RoboDK station: New Station (1).rdk

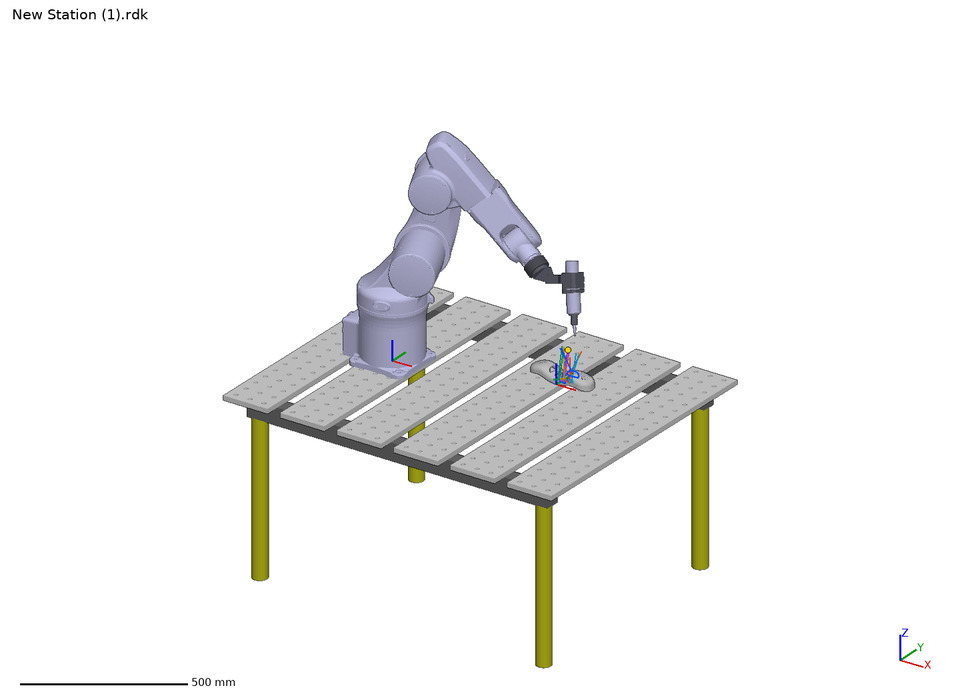
[picture v0: the station drawn from its stored meshes, robots at their saved joint values, targets as dots, program paths as lines]
Station New Station (1). Poses are relative to the parent item; angles as X-Y-Z fixed-axis rotations.
  - frame Adept Viper s650 Base at (-317.82, 0, 0) mm
    - robot Adept Viper s650: 6 axes, payload 5 kg, reach 653 mm, repeatability 0.02 mm, weight 28 kg
        modified DH rows (alpha deg, a mm, theta deg, d mm): 0, 0, 0, 335; -90, 75, 0, 0; 0, 270, -180, 0; -90, 90, 0, 295; 90, 0, 0, 0; -90, 0, 180, 80
        joint limits [-170, -190, -29, -190, -120, -360] to [170, 45, 256, 190, 120, 360]; home [0, -90, 180, 0, 0, 0]; saved at [24.912, -79.024, 220.131, -106.88, 32.598, 110.378]
      - tool Spindle, TCP at (32, 0, 260) mm, rotated rx 0 ry 39 rz 0 deg, size 157.3 x 72 x 259.9 mm
  - object Table at (0, 0, 0) mm, size 1193.8 x 965.2 x 609.6 mm, geometry from welding_table.sld
  - frame Deburring Frame at (278.6, 0, 88) mm
    - object telephone at (0, 0, 0) mm, rotated rx 0 ry 0 rz 90 deg, size 69.7 x 219.4 x 43.4 mm, geometry from telephone.stl
  - machining project telephone Settings: rotZ(0) | rotX(0)*rotY(0) | rotz(0) | onStart | onPathStart | onApproach | onPoint | onRetract | onFinish | SetRPM(%1) | SetTool(%1) | Extruder(%1) | default | default | OutOnMov(%1) | OutOffMov(%1) | onPathFinish | M_RunCode(%1)
  - machining project Path2 settings: rotZ(0) | rotX(0)*rotY(0) | rotz(0) | onStart | onPathStart | onApproach | onPoint | onRetract | onFinish | SetRPM(%1) | SetTool(%1) | Extruder(%1) | default | default | OutOnMov(%1) | OutOffMov(%1) | onPathFinish | M_RunCode(%1)
  - program Path2 (91 instructions, listed below)
  - machining project Path3 settings: rotZ(0) | rotX(0)*rotY(0) | rotz(0) | onStart | onPathStart | onApproach | onPoint | onRetract | onFinish | SetRPM(%1) | SetTool(%1) | Extruder(%1) | default | default | OutOnMov(%1) | OutOffMov(%1) | onPathFinish | M_RunCode(%1)
  - program Path3 (67 instructions, listed below)
  - machining project Path4 settings: rotZ(0) | rotX(0)*rotY(0) | rotz(0) | onStart | onPathStart | onApproach | onPoint | onRetract | onFinish | SetRPM(%1) | SetTool(%1) | Extruder(%1) | default | default | OutOnMov(%1) | OutOffMov(%1) | onPathFinish | M_RunCode(%1)
  - program Path4 (70 instructions, listed below)
  - machining project Path5 settings: rotZ(0) | rotX(0)*rotY(0) | rotz(0) | onStart | onPathStart | onApproach | onPoint | onRetract | onFinish | SetRPM(%1) | SetTool(%1) | Extruder(%1) | default | default | OutOnMov(%1) | OutOffMov(%1) | onPathFinish | M_RunCode(%1)
  - program Path5 (63 instructions, listed below)
  - machining project Path6 settings: rotZ(0) | rotX(0)*rotY(0) | rotz(0) | onStart | onPathStart | onApproach | onPoint | onRetract | onFinish | SetRPM(%1) | SetTool(%1) | Extruder(%1) | default | default | OutOnMov(%1) | OutOffMov(%1) | onPathFinish | M_RunCode(%1)
  - program Path6 (66 instructions, listed below)
  - machining project Path7 settings: rotZ(0) | rotX(0)*rotY(0) | rotz(0) | onStart | onPathStart | onApproach | onPoint | onRetract | onFinish | SetRPM(%1) | SetTool(%1) | Extruder(%1) | default | default | OutOnMov(%1) | OutOffMov(%1) | onPathFinish | M_RunCode(%1)
  - program Path7 (67 instructions, listed below)
  - program telephone (90 instructions, listed below)
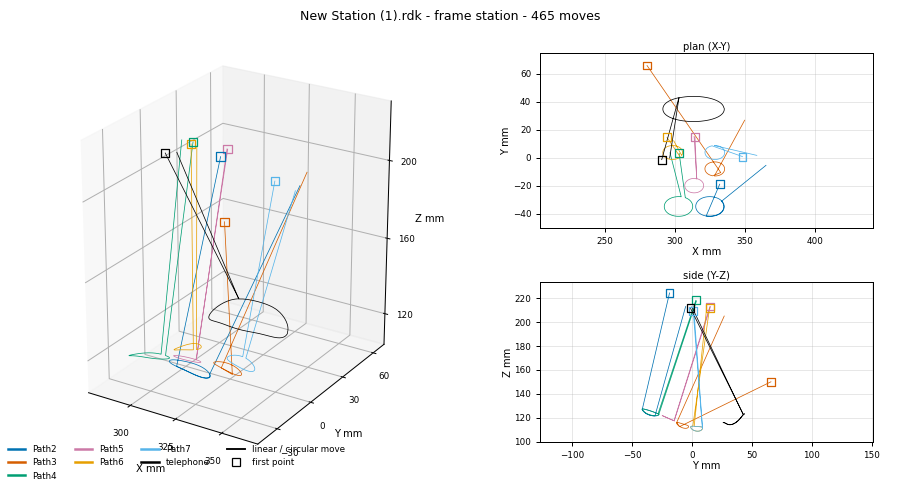
[picture p0: tool path of New Station (1).rdk in frame station, 465 of 465 moves have a stored position in this frame; points joined in program order, loops and branches not executed]

--- program Path2 (robot Adept Viper s650) ---
  Smooth(1)
  Set speed (1000.0 mm/s)
  Set Ref.: Deburring Frame
  Set Tool: Spindle
  Show Spindle
  MoveJ 1 to (53.51, -18.8, 136.35) mm, rotated rx -174.16 ry 13.06 rz 91.32 deg; joints [11.822, -84.058, 219.35, -116.51, 14.318, 120.131]
  MoveL 2 to (53.51, -18.8, 136.35) mm, rotated rx -174.16 ry 13.06 rz 91.32 deg; joints [11.822, -84.058, 219.35, -116.51, 14.318, 120.131]
  MoveL 3 to (43.86, -41.5, 39.44) mm, rotated rx -174.16 ry 13.06 rz 91.32 deg; joints [9.776, -66.741, 219.947, -154.659, 26.957, 158.699]
  MoveL 4 to (43.86, -41.5, 39.44) mm, rotated rx -174.16 ry 13.06 rz 91.32 deg; joints [9.776, -66.741, 219.947, -154.659, 26.957, 158.699]
  Set speed (50.0 mm/s)
  MoveL 5 to (45.33, -41.69, 39.33) mm, rotated rx -172.97 ry 12.9 rz 91.58 deg; joints [10.651, -66.44, 219.515, -151.515, 27.179, 155.489]
  MoveL 6 to (46.59, -41.73, 39.17) mm, rotated rx -170.38 ry 12.62 rz 92.12 deg; joints [12.268, -65.809, 218.773, -145.586, 28.019, 149.205]
  MoveL 7 to (48.09, -41.66, 38.87) mm, rotated rx -167.49 ry 12.41 rz 92.73 deg; joints [14.064, -64.95, 218.023, -139.796, 29.5, 143.03]
  MoveL 8 to (49.56, -41.44, 38.46) mm, rotated rx -164.73 ry 12.23 rz 93.31 deg; joints [15.752, -63.993, 217.309, -135.006, 31.231, 137.876]
  MoveL 9 to (50.68, -41.18, 38.07) mm, rotated rx -162.31 ry 12.13 rz 93.84 deg; joints [17.177, -63.064, 216.743, -131.537, 33, 134.068]
  MoveL 10 to (52.03, -40.71, 37.51) mm, rotated rx -160 ry 12.1 rz 94.36 deg; joints [18.544, -62.081, 216.284, -128.828, 34.916, 131.079]
  MoveL 11 to (53.28, -40.1, 36.89) mm, rotated rx -158.2 ry 12.02 rz 94.76 deg; joints [19.627, -61.249, 215.866, -126.779, 36.409, 128.843]
  MoveL 12 to (53.74, -39.81, 36.63) mm, rotated rx -157.25 ry 11.99 rz 94.98 deg; joints [20.161, -60.808, 215.677, -125.878, 37.231, 127.818]
  MoveL 13 to (54.69, -39.07, 36.05) mm, rotated rx -156.81 ry 12.12 rz 95.14 deg; joints [20.524, -60.571, 215.832, -125.816, 37.899, 127.837]
  MoveL 14 to (55.47, -38.25, 35.52) mm, rotated rx -156.78 ry 12.34 rz 95.24 deg; joints [20.662, -60.55, 216.211, -126.356, 38.326, 128.538]
  MoveL 15 to (55.93, -37.57, 35.15) mm, rotated rx -157.12 ry 12.6 rz 95.26 deg; joints [20.578, -60.709, 216.714, -127.342, 38.499, 129.714]
  MoveL 16 to (56.35, -36.71, 34.75) mm, rotated rx -157.66 ry 12.9 rz 95.24 deg; joints [20.401, -60.973, 217.335, -128.582, 38.581, 131.196]
  MoveL 17 to (56.4, -36.58, 34.7) mm, rotated rx -158.04 ry 13.08 rz 95.22 deg; joints [20.221, -61.139, 217.652, -129.392, 38.555, 132.109]
  MoveL 18 to (56.62, -35.75, 34.39) mm, rotated rx -158.41 ry 13.23 rz 95.18 deg; joints [20.104, -61.343, 218.07, -130.132, 38.577, 133.023]
  MoveL 19 to (56.71, -34.89, 34.12) mm, rotated rx -159.01 ry 13.46 rz 95.1 deg; joints [19.853, -61.655, 218.636, -131.298, 38.533, 134.398]
  MoveL 20 to (56.68, -34.23, 33.95) mm, rotated rx -159.47 ry 13.6 rz 95.03 deg; joints [19.65, -61.902, 219.035, -132.122, 38.457, 135.366]
  MoveL 21 to (56.63, -33.9, 33.88) mm, rotated rx -159.71 ry 13.68 rz 95 deg; joints [19.537, -62.031, 219.25, -132.577, 38.428, 135.892]
  MoveL 22 to (56.44, -33.13, 33.73) mm, rotated rx -159.89 ry 13.75 rz 94.97 deg; joints [19.455, -62.189, 219.552, -133.002, 38.469, 136.39]
  MoveL 23 to (56.13, -32.37, 33.63) mm, rotated rx -160.06 ry 13.79 rz 94.94 deg; joints [19.365, -62.356, 219.834, -133.373, 38.48, 136.815]
  MoveL 24 to (56.07, -32.27, 33.62) mm, rotated rx -160.12 ry 13.83 rz 94.94 deg; joints [19.327, -62.396, 219.921, -133.552, 38.502, 137.012]
  MoveL 25 to (55.61, -31.52, 33.57) mm, rotated rx -160.19 ry 13.93 rz 94.96 deg; joints [19.262, -62.53, 220.248, -133.964, 38.66, 137.442]
  MoveL 26 to (55, -30.79, 33.58) mm, rotated rx -160.3 ry 14.06 rz 94.97 deg; joints [19.152, -62.691, 220.623, -134.513, 38.828, 137.999]
  MoveL 27 to (54.88, -30.66, 33.59) mm, rotated rx -160.47 ry 14.24 rz 94.99 deg; joints [19.047, -62.763, 220.887, -135.12, 38.995, 138.642]
  MoveL 28 to (54.02, -29.92, 33.67) mm, rotated rx -160.96 ry 14.61 rz 94.98 deg; joints [18.699, -63.064, 221.608, -136.63, 39.279, 140.214]
  MoveL 29 to (53.03, -29.28, 33.8) mm, rotated rx -161.94 ry 15.12 rz 94.86 deg; joints [18.069, -63.52, 222.542, -138.962, 39.476, 142.68]
  MoveL 30 to (52.23, -28.87, 33.92) mm, rotated rx -163.91 ry 15.86 rz 94.51 deg; joints [16.933, -64.207, 223.779, -142.808, 39.497, 146.856]
  MoveL 31 to (50.89, -28.36, 34.12) mm, rotated rx -166.32 ry 16.57 rz 93.97 deg; joints [15.492, -64.991, 225.06, -147.237, 39.413, 151.619]
  MoveL 32 to (49.47, -27.98, 34.33) mm, rotated rx -168.54 ry 17.08 rz 93.41 deg; joints [14.119, -65.637, 226.045, -151.185, 39.278, 155.822]
  MoveL 33 to (48.32, -27.79, 34.5) mm, rotated rx -170.84 ry 17.46 rz 92.77 deg; joints [12.719, -66.194, 226.83, -155.099, 39.06, 160.014]
  MoveL 34 to (46.67, -27.67, 34.72) mm, rotated rx -172.86 ry 17.76 rz 92.19 deg; joints [11.384, -66.632, 227.471, -158.665, 38.953, 163.726]
  MoveL 35 to (45, -27.73, 34.92) mm, rotated rx -174.72 ry 17.95 rz 91.63 deg; joints [10.113, -66.972, 227.927, -161.947, 38.808, 167.106]
  MoveL 36 to (43.78, -27.89, 35.08) mm, rotated rx -175.97 ry 18.12 rz 91.25 deg; joints [9.236, -67.133, 228.219, -164.217, 38.847, 169.427]
  MoveL 37 to (42.27, -28.24, 35.29) mm, rotated rx -176.64 ry 18.23 rz 91.05 deg; joints [8.625, -67.201, 228.359, -165.629, 38.902, 170.747]
  MoveL 38 to (40.89, -28.75, 35.53) mm, rotated rx -176.95 ry 18.33 rz 90.96 deg; joints [8.228, -67.202, 228.406, -166.445, 38.983, 171.424]
  MoveL 39 to (40.41, -28.98, 35.63) mm, rotated rx -176.9 ry 18.46 rz 90.98 deg; joints [8.178, -67.138, 228.477, -166.546, 39.248, 171.458]
  MoveL 40 to (39.33, -29.62, 35.89) mm, rotated rx -176.68 ry 18.53 rz 91.06 deg; joints [8.118, -67.068, 228.403, -166.466, 39.328, 171.186]
  MoveL 41 to (38.41, -30.35, 36.19) mm, rotated rx -176.39 ry 18.62 rz 91.15 deg; joints [8.116, -66.969, 228.315, -166.271, 39.458, 170.807]
  MoveL 42 to (37.75, -31.04, 36.46) mm, rotated rx -176.1 ry 18.66 rz 91.25 deg; joints [8.158, -66.887, 228.182, -165.98, 39.479, 170.362]
  MoveL 43 to (37.17, -31.88, 36.78) mm, rotated rx -175.9 ry 18.66 rz 91.31 deg; joints [8.155, -66.817, 227.997, -165.796, 39.392, 170.041]
  MoveL 44 to (36.78, -32.66, 37.08) mm, rotated rx -175.77 ry 18.64 rz 91.35 deg; joints [8.146, -66.765, 227.798, -165.657, 39.238, 169.804]
  MoveL 45 to (36.52, -33.55, 37.4) mm, rotated rx -175.73 ry 18.58 rz 91.36 deg; joints [8.107, -66.726, 227.548, -165.591, 38.975, 169.662]
  MoveL 46 to (36.49, -33.71, 37.46) mm, rotated rx -175.79 ry 18.46 rz 91.34 deg; joints [8.064, -66.767, 227.422, -165.611, 38.691, 169.675]
  MoveL 47 to (36.4, -34.56, 37.75) mm, rotated rx -175.86 ry 18.36 rz 91.31 deg; joints [7.995, -66.754, 227.145, -165.641, 38.319, 169.671]
  MoveL 48 to (36.44, -35.26, 37.98) mm, rotated rx -175.93 ry 18.22 rz 91.27 deg; joints [7.945, -66.757, 226.875, -165.64, 37.909, 169.657]
  MoveL 49 to (36.47, -35.43, 38.03) mm, rotated rx -176.04 ry 18.04 rz 91.23 deg; joints [7.883, -66.824, 226.687, -165.674, 37.464, 169.694]
  MoveL 50 to (36.55, -35.87, 38.17) mm, rotated rx -176.16 ry 17.8 rz 91.18 deg; joints [7.816, -66.884, 226.382, -165.673, 36.854, 169.695]
  MoveL 51 to (36.82, -36.7, 38.42) mm, rotated rx -176.39 ry 17.5 rz 91.09 deg; joints [7.705, -66.933, 225.94, -165.772, 36.048, 169.825]
  MoveL 52 to (37.24, -37.52, 38.65) mm, rotated rx -176.52 ry 17.21 rz 91.03 deg; joints [7.676, -66.954, 225.493, -165.673, 35.297, 169.756]
  MoveL 53 to (37.33, -37.66, 38.69) mm, rotated rx -176.89 ry 16.75 rz 90.9 deg; joints [7.471, -67.114, 225.075, -165.954, 34.228, 170.077]
  MoveL 54 to (37.95, -38.47, 38.91) mm, rotated rx -177.09 ry 16.38 rz 90.82 deg; joints [7.424, -67.143, 224.535, -165.89, 33.278, 170.077]
  MoveL 55 to (38.7, -39.22, 39.09) mm, rotated rx -177.32 ry 15.94 rz 90.74 deg; joints [7.382, -67.179, 223.946, -165.795, 32.213, 170.065]
  MoveL 56 to (39.08, -39.52, 39.16) mm, rotated rx -177.53 ry 15.3 rz 90.65 deg; joints [7.288, -67.295, 223.269, -165.625, 30.785, 169.925]
  MoveL 57 to (40.1, -40.19, 39.3) mm, rotated rx -177.34 ry 14.81 rz 90.68 deg; joints [7.513, -67.265, 222.578, -164.583, 29.711, 168.919]
  MoveL 58 to (41.24, -40.74, 39.4) mm, rotated rx -176.81 ry 14.17 rz 90.78 deg; joints [7.947, -67.204, 221.704, -162.55, 28.426, 166.864]
  MoveL 59 to (42.44, -41.17, 39.45) mm, rotated rx -175.65 ry 13.56 rz 91.02 deg; joints [8.749, -67.031, 220.797, -159.011, 27.45, 163.202]
  MoveL 60 to (43.86, -41.5, 39.44) mm, rotated rx -173.92 ry 13.08 rz 91.38 deg; joints [9.914, -66.696, 219.942, -154.19, 27.101, 158.188]
  MoveL 61 to (45.34, -41.52, 39.29) mm, rotated rx -171.6 ry 12.58 rz 91.84 deg; joints [11.422, -66.186, 219.018, -148.104, 27.266, 151.813]
  MoveL 62 to (46.58, -41.56, 39.13) mm, rotated rx -168.9 ry 12.22 rz 92.38 deg; joints [13.088, -65.46, 218.138, -141.952, 28.204, 145.277]
  MoveL 63 to (48.06, -41.49, 38.83) mm, rotated rx -166.24 ry 11.93 rz 92.9 deg; joints [14.75, -64.594, 217.31, -136.578, 29.594, 139.553]
  MoveL 64 to (49.51, -41.27, 38.43) mm, rotated rx -163.53 ry 11.65 rz 93.42 deg; joints [16.398, -63.592, 216.465, -131.819, 31.279, 134.431]
  MoveL 65 to (50.62, -41, 38.05) mm, rotated rx -161.08 ry 11.6 rz 93.94 deg; joints [17.825, -62.605, 215.925, -128.66, 33.238, 130.925]
  MoveL 66 to (51.95, -40.53, 37.5) mm, rotated rx -159.3 ry 11.65 rz 94.36 deg; joints [18.915, -61.802, 215.641, -126.857, 34.889, 128.946]
  MoveL 67 to (53.17, -39.92, 36.89) mm, rotated rx -157.83 ry 11.77 rz 94.75 deg; joints [19.816, -61.109, 215.54, -125.785, 36.408, 127.762]
  MoveL 68 to (53.63, -39.64, 36.64) mm, rotated rx -157.19 ry 12.16 rz 95.06 deg; joints [20.172, -60.818, 215.916, -126.318, 37.502, 128.254]
  MoveL 69 to (54.55, -38.91, 36.07) mm, rotated rx -157.07 ry 12.45 rz 95.21 deg; joints [20.369, -60.726, 216.335, -126.963, 38.124, 129.049]
  MoveL 70 to (55.3, -38.1, 35.55) mm, rotated rx -157.35 ry 12.89 rz 95.32 deg; joints [20.343, -60.835, 217.027, -128.315, 38.604, 130.633]
  MoveL 71 to (55.75, -37.44, 35.19) mm, rotated rx -157.59 ry 13.07 rz 95.33 deg; joints [20.309, -60.941, 217.398, -128.977, 38.761, 131.455]
  MoveL 72 to (56.15, -36.6, 34.8) mm, rotated rx -158.25 ry 13.39 rz 95.28 deg; joints [20.064, -61.246, 218.061, -130.387, 38.805, 133.132]
  MoveL 73 to (56.19, -36.48, 34.75) mm, rotated rx -158.63 ry 13.46 rz 95.21 deg; joints [19.891, -61.408, 218.241, -130.907, 38.632, 133.747]
  MoveL 74 to (56.4, -35.68, 34.45) mm, rotated rx -159.14 ry 13.62 rz 95.13 deg; joints [19.698, -61.665, 218.69, -131.811, 38.568, 134.849]
  MoveL 75 to (56.47, -34.86, 34.2) mm, rotated rx -159.52 ry 13.7 rz 95.05 deg; joints [19.559, -61.883, 219.034, -132.412, 38.492, 135.601]
  MoveL 76 to (56.44, -34.23, 34.04) mm, rotated rx -159.82 ry 13.74 rz 94.99 deg; joints [19.439, -62.062, 219.279, -132.837, 38.392, 136.129]
  MoveL 77 to (56.4, -33.92, 33.96) mm, rotated rx -159.94 ry 13.76 rz 94.96 deg; joints [19.387, -62.143, 219.405, -133.043, 38.37, 136.378]
  MoveL 78 to (56.21, -33.19, 33.83) mm, rotated rx -160.06 ry 13.79 rz 94.94 deg; joints [19.335, -62.276, 219.638, -133.302, 38.388, 136.694]
  MoveL 79 to (55.91, -32.47, 33.73) mm, rotated rx -160.13 ry 13.82 rz 94.94 deg; joints [19.294, -62.398, 219.877, -133.542, 38.452, 136.967]
  MoveL 80 to (55.86, -32.37, 33.72) mm, rotated rx -160.19 ry 13.91 rz 94.95 deg; joints [19.258, -62.429, 220.008, -133.814, 38.546, 137.257]
  MoveL 81 to (55.42, -31.65, 33.68) mm, rotated rx -160.15 ry 13.86 rz 94.94 deg; joints [19.251, -62.532, 220.147, -133.779, 38.549, 137.212]
  MoveL 82 to (54.83, -30.95, 33.69) mm, rotated rx -160.25 ry 14 rz 94.96 deg; joints [19.147, -62.684, 220.52, -134.331, 38.732, 137.772]
  Set speed (1000.0 mm/s)
  MoveL 83 to (54.83, -30.95, 33.69) mm, rotated rx -160.25 ry 14 rz 94.96 deg; joints [19.147, -62.684, 220.52, -134.331, 38.732, 137.772]
  MoveL 84 to (86.53, -5.35, 125.01) mm, rotated rx -160.25 ry 14 rz 94.96 deg; joints [24.912, -79.024, 220.131, -106.88, 32.598, 110.378]

--- program Path3 (robot Adept Viper s650) ---
  Smooth(1)
  Set speed (1000.0 mm/s)
  Set Ref.: Deburring Frame
  Set Tool: Spindle
  Show Spindle
  MoveJ 1 to (1.67, 65.89, 62.11) mm, rotated rx 112.25 ry 7.94 rz 37.78 deg; joints [0.056, -47.226, 255.354, -174.919, 106.228, -108.091]
  MoveL 2 to (1.67, 65.89, 62.11) mm, rotated rx 112.25 ry 7.94 rz 37.78 deg; joints [0.056, -47.226, 255.354, -174.919, 106.228, -108.091]
  MoveL 3 to (54.24, -10.47, 24.61) mm, rotated rx 114.73 ry 26.32 rz 46.09 deg; joints [4.762, -22.597, 229.967, -175.784, 116.598, -123.556]
  MoveL 4 to (54.24, -10.47, 24.61) mm, rotated rx 114.73 ry 26.32 rz 46.09 deg; joints [4.762, -22.597, 229.967, -175.784, 116.598, -123.556]
  Set speed (50.0 mm/s)
  MoveL 5 to (48.57, -12.8, 28.08) mm, rotated rx 159.78 ry 39.33 rz 76.86 deg; joints [5.018, -40.691, 237.454, -177.659, 97.243, -163.59]
  MoveL 6 to (47.94, -12.67, 28.14) mm, rotated rx -169.03 ry 22.67 rz 94.27 deg; joints [14.025, -63.487, 233.835, -158.545, 53.468, -195.376]
  MoveL 7 to (46.89, -12.37, 28.19) mm, rotated rx -170.53 ry 22.4 rz 93.64 deg; joints [13.125, -64.139, 233.981, -160.07, 52.42, -193.816]
  MoveL 8 to (45.93, -11.96, 28.15) mm, rotated rx -171.82 ry 22.21 rz 93.11 deg; joints [12.327, -64.636, 234.159, -161.496, 51.69, -192.362]
  MoveL 9 to (45.4, -11.66, 28.09) mm, rotated rx -172.72 ry 21.92 rz 92.73 deg; joints [11.785, -65.072, 234.167, -162.404, 50.838, -191.437]
  MoveL 10 to (44.66, -11.13, 27.96) mm, rotated rx -173.43 ry 21.4 rz 92.41 deg; joints [11.309, -65.625, 234.055, -163.035, 49.58, -190.865]
  MoveL 11 to (44.05, -10.53, 27.79) mm, rotated rx -173.69 ry 21.02 rz 92.27 deg; joints [11.086, -65.986, 233.978, -163.23, 48.738, -190.746]
  MoveL 12 to (43.98, -10.45, 27.76) mm, rotated rx -173.82 ry 20.62 rz 92.18 deg; joints [11.001, -66.278, 233.741, -163.162, 47.822, -190.853]
  MoveL 13 to (43.54, -9.83, 27.58) mm, rotated rx -173.99 ry 19.92 rz 92.06 deg; joints [10.851, -66.801, 233.402, -163.006, 46.272, -191.11]
  MoveL 14 to (43.23, -9.2, 27.38) mm, rotated rx -173.95 ry 19.13 rz 91.99 deg; joints [10.829, -67.302, 232.956, -162.489, 44.597, -191.739]
  MoveL 15 to (43.12, -8.87, 27.28) mm, rotated rx -173.82 ry 18.39 rz 91.96 deg; joints [10.883, -67.702, 232.44, -161.795, 43.026, -192.532]
  MoveL 16 to (43, -8.29, 27.1) mm, rotated rx -173.76 ry 17.72 rz 91.91 deg; joints [10.901, -68.066, 232.024, -161.223, 41.643, -193.173]
  MoveL 17 to (42.99, -8.22, 27.08) mm, rotated rx -173.72 ry 17.09 rz 91.85 deg; joints [10.914, -68.35, 231.513, -160.634, 40.291, -193.832]
  MoveL 18 to (42.97, -7.57, 26.89) mm, rotated rx -173.66 ry 16.35 rz 91.79 deg; joints [10.954, -68.699, 231.002, -159.866, 38.769, -194.658]
  MoveL 19 to (43, -7.34, 26.82) mm, rotated rx -173.54 ry 15.47 rz 91.73 deg; joints [11.013, -69.014, 230.257, -158.807, 36.96, -195.804]
  MoveL 20 to (43.14, -6.69, 26.62) mm, rotated rx -173.44 ry 14.52 rz 91.65 deg; joints [11.092, -69.343, 229.503, -157.566, 35.068, -197.1]
  MoveL 21 to (43.26, -6.34, 26.52) mm, rotated rx -173.43 ry 13.67 rz 91.56 deg; joints [11.105, -69.589, 228.762, -156.484, 33.356, -198.232]
  MoveL 22 to (43.42, -6.01, 26.42) mm, rotated rx -173.23 ry 12.74 rz 91.5 deg; joints [11.231, -69.768, 227.887, -154.819, 31.582, -199.964]
  MoveL 23 to (43.83, -5.37, 26.23) mm, rotated rx -172.99 ry 11.59 rz 91.42 deg; joints [11.426, -69.939, 226.791, -152.439, 29.459, -202.387]
  MoveL 24 to (44.3, -4.85, 26.08) mm, rotated rx -172.66 ry 10.38 rz 91.33 deg; joints [11.673, -70.003, 225.556, -149.424, 27.361, -205.452]
  MoveL 25 to (45.04, -4.25, 25.87) mm, rotated rx -172.01 ry 9.21 rz 91.29 deg; joints [12.166, -69.908, 224.264, -145.251, 25.634, -209.656]
  MoveL 26 to (46, -3.7, 25.65) mm, rotated rx -170.97 ry 8.3 rz 91.31 deg; joints [12.945, -69.621, 223.122, -140.355, 24.772, -214.564]
  MoveL 27 to (47.09, -3.29, 25.4) mm, rotated rx -169.51 ry 7.77 rz 91.43 deg; joints [14.016, -69.147, 222.263, -135.475, 25.003, -219.447]
  MoveL 28 to (48.28, -3.01, 25.13) mm, rotated rx -168.12 ry 7.6 rz 91.59 deg; joints [15.066, -68.635, 221.773, -132.011, 25.886, -222.878]
  MoveL 29 to (48.69, -2.95, 25.03) mm, rotated rx -166.9 ry 7.58 rz 91.76 deg; joints [15.877, -68.19, 221.477, -129.723, 26.848, -225.215]
  MoveL 30 to (49.99, -2.87, 24.7) mm, rotated rx -165.32 ry 7.68 rz 92.01 deg; joints [17.032, -67.511, 221.164, -127.27, 28.358, -227.631]
  MoveL 31 to (51.3, -2.96, 24.36) mm, rotated rx -163.86 ry 7.75 rz 92.23 deg; joints [18.081, -66.804, 220.793, -125.187, 29.751, -229.681]
  MoveL 32 to (51.51, -2.99, 24.3) mm, rotated rx -162.89 ry 7.95 rz 92.44 deg; joints [18.688, -66.388, 220.771, -124.486, 30.853, -230.431]
  MoveL 33 to (52.65, -3.23, 23.98) mm, rotated rx -161.8 ry 8.4 rz 92.75 deg; joints [19.468, -65.805, 220.907, -124.353, 32.414, -230.505]
  MoveL 34 to (53.7, -3.6, 23.69) mm, rotated rx -160.98 ry 8.89 rz 93.05 deg; joints [20.071, -65.303, 221.113, -124.641, 33.782, -230.153]
  MoveL 35 to (54.6, -4.06, 23.46) mm, rotated rx -160.88 ry 9.51 rz 93.28 deg; joints [20.231, -65.126, 221.659, -126.158, 34.719, -228.513]
  MoveL 36 to (55.29, -4.55, 23.32) mm, rotated rx -161.28 ry 10.32 rz 93.47 deg; joints [20.082, -65.172, 222.532, -128.668, 35.524, -225.839]
  MoveL 37 to (55.85, -5.07, 23.25) mm, rotated rx -161.89 ry 11.28 rz 93.66 deg; joints [19.794, -65.273, 223.605, -131.718, 36.473, -222.604]
  MoveL 38 to (56.26, -5.59, 23.24) mm, rotated rx -162.44 ry 12.21 rz 93.83 deg; joints [19.517, -65.315, 224.598, -134.473, 37.506, -219.687]
  MoveL 39 to (56.43, -5.85, 23.25) mm, rotated rx -162.79 ry 12.91 rz 93.96 deg; joints [19.325, -65.315, 225.357, -136.425, 38.407, -217.623]
  MoveL 40 to (56.58, -6.14, 23.28) mm, rotated rx -163.04 ry 13.52 rz 94.08 deg; joints [19.188, -65.26, 225.969, -137.968, 39.257, -215.992]
  MoveL 41 to (56.72, -6.44, 23.32) mm, rotated rx -163.24 ry 14.15 rz 94.21 deg; joints [19.068, -65.164, 226.573, -139.433, 40.195, -214.442]
  MoveL 42 to (56.82, -6.72, 23.37) mm, rotated rx -163.39 ry 14.76 rz 94.35 deg; joints [18.974, -65.031, 227.139, -140.743, 41.17, -213.057]
  MoveL 43 to (56.9, -7.01, 23.43) mm, rotated rx -163.49 ry 15.5 rz 94.53 deg; joints [18.894, -64.824, 227.799, -142.166, 42.424, -211.552]
  MoveL 44 to (57, -7.59, 23.59) mm, rotated rx -163.51 ry 16.29 rz 94.75 deg; joints [18.841, -64.511, 228.408, -143.494, 43.829, -210.165]
  MoveL 45 to (57.01, -7.75, 23.64) mm, rotated rx -163.42 ry 16.99 rz 94.97 deg; joints [18.85, -64.196, 228.988, -144.521, 45.2, -209.08]
  MoveL 46 to (56.99, -8.37, 23.85) mm, rotated rx -163.16 ry 17.86 rz 95.3 deg; joints [18.902, -63.694, 229.564, -145.553, 46.938, -208.031]
  MoveL 47 to (56.85, -9.04, 24.13) mm, rotated rx -162.67 ry 18.83 rz 95.75 deg; joints [19.031, -63.017, 230.154, -146.464, 49.031, -207.148]
  MoveL 48 to (56.6, -9.7, 24.46) mm, rotated rx -162.18 ry 19.49 rz 96.12 deg; joints [19.143, -62.477, 230.489, -146.953, 50.528, -206.742]
  MoveL 49 to (56.56, -9.79, 24.51) mm, rotated rx -161.62 ry 20.09 rz 96.51 deg; joints [19.35, -61.916, 230.84, -147.241, 52.027, -206.476]
  MoveL 50 to (56.1, -10.5, 24.94) mm, rotated rx -161.02 ry 20.74 rz 96.94 deg; joints [19.451, -61.321, 231.121, -147.636, 53.544, -206.229]
  MoveL 51 to (55.46, -11.18, 25.43) mm, rotated rx -160.7 ry 21.29 rz 97.25 deg; joints [19.398, -60.9, 231.391, -148.169, 54.729, -205.847]
  MoveL 52 to (54.66, -11.77, 25.95) mm, rotated rx -160.62 ry 21.61 rz 97.38 deg; joints [19.235, -60.746, 231.558, -148.628, 55.302, -205.548]
  MoveL 53 to (53.72, -12.25, 26.47) mm, rotated rx -161.03 ry 22.06 rz 97.35 deg; joints [18.817, -60.714, 231.923, -149.656, 55.898, -204.6]
  MoveL 54 to (53.41, -12.37, 26.62) mm, rotated rx -161.92 ry 22.24 rz 97.04 deg; joints [18.339, -60.967, 232.194, -150.654, 55.799, -203.501]
  MoveL 55 to (52.32, -12.69, 27.11) mm, rotated rx -162.84 ry 22.5 rz 96.74 deg; joints [17.701, -61.25, 232.532, -151.886, 55.789, -202.298]
  MoveL 56 to (51.16, -12.88, 27.51) mm, rotated rx -164.13 ry 22.67 rz 96.25 deg; joints [16.891, -61.704, 232.893, -153.378, 55.481, -200.782]
  MoveL 57 to (50.87, -12.9, 27.6) mm, rotated rx -164.12 ry 22.66 rz 96.26 deg; joints [16.852, -61.736, 232.898, -153.399, 55.445, -200.812]
  MoveL 58 to (49.71, -12.91, 27.88) mm, rotated rx -165.2 ry 22.75 rz 95.84 deg; joints [16.152, -62.142, 233.192, -154.643, 55.121, -199.573]
  Set speed (1000.0 mm/s)
  MoveL 59 to (49.71, -12.91, 27.88) mm, rotated rx -165.2 ry 22.75 rz 95.84 deg; joints [16.152, -62.142, 233.192, -154.643, 55.121, -199.573]
  MoveL 60 to (71.33, 26.88, 117.04) mm, rotated rx -165.2 ry 22.75 rz 95.84 deg; joints [22.134, -87.144, 239.403, -137.89, 40.446, -215.747]

--- program Path4 (robot Adept Viper s650) ---
  Smooth(1)
  Set speed (1000.0 mm/s)
  Set Ref.: Deburring Frame
  Set Tool: Spindle
  Show Spindle
  MoveJ 1 to (24.58, 3.18, 130.16) mm, rotated rx 177.2 ry 18.39 rz 89.12 deg; joints [2.623, -90.691, 232.668, -177.654, 19.439, -178.563]
  MoveL 2 to (24.58, 3.18, 130.16) mm, rotated rx 177.2 ry 18.39 rz 89.12 deg; joints [2.623, -90.691, 232.668, -177.654, 19.439, -178.563]
  MoveL 3 to (28.97, -28.41, 35.38) mm, rotated rx 177.2 ry 18.39 rz 89.12 deg; joints [3.097, -67.668, 229.265, -178.127, 39.054, -177.55]
  MoveL 4 to (28.97, -28.41, 35.38) mm, rotated rx 177.2 ry 18.39 rz 89.12 deg; joints [3.097, -67.668, 229.265, -178.127, 39.054, -177.55]
  Set speed (50.0 mm/s)
  MoveL 5 to (28.97, -28.41, 35.38) mm, rotated rx 177.29 ry 18.37 rz 89.15 deg; joints [3.145, -67.678, 229.242, -177.989, 38.996, -177.703]
  MoveL 6 to (29.14, -28.47, 35.41) mm, rotated rx 177.38 ry 18.36 rz 89.17 deg; joints [3.22, -67.678, 229.216, -177.815, 38.961, -177.87]
  MoveL 7 to (30.31, -28.98, 35.63) mm, rotated rx 177.23 ry 18.38 rz 89.13 deg; joints [3.323, -67.631, 229.104, -177.792, 38.918, -177.717]
  MoveL 8 to (31.36, -29.61, 35.89) mm, rotated rx 176.94 ry 18.42 rz 89.03 deg; joints [3.324, -67.561, 229.002, -178.028, 38.943, -177.297]
  MoveL 9 to (31.77, -29.91, 36.01) mm, rotated rx 176.61 ry 18.47 rz 88.93 deg; joints [3.212, -67.511, 228.989, -178.436, 39.044, -176.781]
  MoveL 10 to (32.57, -30.63, 36.3) mm, rotated rx 176.26 ry 18.52 rz 88.81 deg; joints [3.142, -67.432, 228.874, -178.807, 39.071, -176.249]
  MoveL 11 to (33.23, -31.43, 36.62) mm, rotated rx 176.02 ry 18.6 rz 88.73 deg; joints [3.114, -67.332, 228.766, -179.028, 39.16, -175.899]
  MoveL 12 to (33.37, -31.64, 36.7) mm, rotated rx 175.87 ry 18.64 rz 88.68 deg; joints [3.059, -67.294, 228.76, -179.213, 39.241, -175.67]
  MoveL 13 to (33.81, -32.47, 37.01) mm, rotated rx 175.75 ry 18.65 rz 88.64 deg; joints [3.056, -67.228, 228.577, -179.312, 39.137, -175.497]
  MoveL 14 to (34.1, -33.32, 37.32) mm, rotated rx 175.71 ry 18.64 rz 88.63 deg; joints [3.074, -67.166, 228.377, -179.317, 38.996, -175.455]
  MoveL 15 to (34.13, -33.45, 37.36) mm, rotated rx 175.74 ry 18.6 rz 88.64 deg; joints [3.092, -67.175, 228.312, -179.27, 38.88, -175.508]
  MoveL 16 to (34.25, -34.3, 37.66) mm, rotated rx 175.78 ry 18.49 rz 88.66 deg; joints [3.115, -67.157, 228.019, -179.218, 38.491, -175.57]
  MoveL 17 to (34.24, -35.07, 37.91) mm, rotated rx 175.87 ry 18.35 rz 88.7 deg; joints [3.139, -67.155, 227.721, -179.131, 38.052, -175.692]
  MoveL 18 to (34.23, -35.14, 37.94) mm, rotated rx 175.98 ry 18.27 rz 88.74 deg; joints [3.191, -67.186, 227.625, -178.976, 37.833, -175.876]
  MoveL 19 to (34.2, -35.42, 38.03) mm, rotated rx 176.17 ry 18.12 rz 88.81 deg; joints [3.273, -67.224, 227.421, -178.717, 37.432, -176.189]
  MoveL 20 to (33.99, -36.29, 38.3) mm, rotated rx 176.51 ry 17.77 rz 88.93 deg; joints [3.386, -67.287, 226.9, -178.29, 36.481, -176.741]
  MoveL 21 to (33.61, -37.18, 38.56) mm, rotated rx 176.88 ry 17.25 rz 89.08 deg; joints [3.482, -67.389, 226.218, -177.835, 35.162, -177.364]
  MoveL 22 to (33.07, -38.02, 38.79) mm, rotated rx 177.23 ry 16.67 rz 89.2 deg; joints [3.537, -67.489, 225.483, -177.429, 33.739, -177.953]
  MoveL 23 to (32.48, -38.71, 38.97) mm, rotated rx 177.58 ry 16.03 rz 89.33 deg; joints [3.589, -67.591, 224.713, -176.98, 32.221, -178.594]
  MoveL 24 to (31.61, -39.48, 39.15) mm, rotated rx 177.93 ry 15.34 rz 89.45 deg; joints [3.599, -67.667, 223.862, -176.54, 30.599, -179.257]
  MoveL 25 to (30.6, -40.15, 39.3) mm, rotated rx 178.08 ry 14.88 rz 89.51 deg; joints [3.496, -67.684, 223.258, -176.487, 29.514, -179.496]
  MoveL 26 to (30.23, -40.35, 39.34) mm, rotated rx 178.07 ry 14.49 rz 89.52 deg; joints [3.411, -67.729, 222.822, -176.593, 28.638, -179.462]
  MoveL 27 to (28.94, -40.91, 39.44) mm, rotated rx 177.76 ry 13.96 rz 89.46 deg; joints [3.003, -67.746, 222.191, -177.638, 27.46, -178.553]
  MoveL 28 to (27.54, -41.33, 39.48) mm, rotated rx 176.95 ry 13.55 rz 89.29 deg; joints [2.3, -67.743, 221.728, -179.937, 26.61, -176.307]
  MoveL 29 to (26.57, -41.52, 39.47) mm, rotated rx 175.7 ry 13.21 rz 89.01 deg; joints [1.402, -67.719, 221.396, -183.314, 26.061, -172.85]
  MoveL 30 to (25.06, -41.68, 39.38) mm, rotated rx 173.69 ry 12.83 rz 88.59 deg; joints [-0.018, -67.599, 221.049, -188.777, 25.782, -167.246]
  MoveL 31 to (23.55, -41.7, 39.18) mm, rotated rx 167.47 ry 8.8 rz 68.08 deg; joints [7.356, -66.971, 217.081, -144.87, 21.817, -185.807]
  MoveL 32 to (22.59, -41.63, 39) mm, rotated rx 165.66 ry 8.09 rz 67.81 deg; joints [6.065, -67.259, 217.358, -150.335, 20.779, -180.119]
  MoveL 33 to (22.08, -41.57, 38.89) mm, rotated rx 163.87 ry 9.39 rz 67.17 deg; joints [5.645, -67.396, 219.529, -156.152, 23.991, -173.393]
  MoveL 34 to (21.1, -41.41, 38.63) mm, rotated rx 162.14 ry 8.45 rz 66.95 deg; joints [4.294, -67.587, 219.538, -161.414, 22.926, -168]
  MoveL 35 to (19.69, -41.05, 38.17) mm, rotated rx 160.42 ry 5.66 rz 67.24 deg; joints [2.11, -67.656, 217.689, -169.528, 18.437, -160.422]
  MoveL 36 to (18.63, -40.66, 37.75) mm, rotated rx 158.38 ry 4.96 rz 67.01 deg; joints [0.674, -67.652, 218.03, -177.395, 18.683, -152.279]
  MoveL 37 to (17.48, -40.1, 37.21) mm, rotated rx 156.61 ry 4.47 rz 66.78 deg; joints [-0.559, -67.592, 218.471, -183.707, 19.443, -145.719]
  MoveL 38 to (16.47, -39.44, 36.66) mm, rotated rx 155.34 ry 4.35 rz 66.53 deg; joints [-1.365, -67.542, 219.099, -187.205, 20.627, -141.981]
  MoveL 39 to (15.61, -38.67, 36.11) mm, rotated rx 154.76 ry 4.46 rz 66.36 deg; joints [-1.713, -67.546, 219.663, -188.235, 21.563, -140.837]
  MoveL 40 to (15.45, -38.5, 36) mm, rotated rx 154.67 ry 4.68 rz 66.25 deg; joints [-1.678, -67.564, 219.985, -187.774, 22.093, -141.208]
  MoveL 41 to (14.85, -37.71, 35.55) mm, rotated rx 154.88 ry 5.1 rz 66.15 deg; joints [-1.483, -67.653, 220.535, -186.33, 22.807, -142.639]
  MoveL 42 to (14.35, -36.77, 35.1) mm, rotated rx 155.28 ry 5.55 rz 66.09 deg; joints [-1.171, -67.772, 221.052, -184.517, 23.4, -144.478]
  MoveL 43 to (14.1, -35.96, 34.78) mm, rotated rx 155.73 ry 5.9 rz 66.08 deg; joints [-0.842, -67.884, 221.406, -182.855, 23.745, -146.188]
  MoveL 44 to (13.97, -35.16, 34.51) mm, rotated rx 156.07 ry 6.13 rz 66.09 deg; joints [-0.598, -67.99, 221.682, -181.681, 23.973, -147.402]
  MoveL 45 to (13.96, -34.7, 34.38) mm, rotated rx 156.35 ry 6.3 rz 66.11 deg; joints [-0.388, -68.058, 221.843, -180.734, 24.105, -148.377]
  MoveL 46 to (14.03, -33.91, 34.18) mm, rotated rx 156.64 ry 6.48 rz 66.12 deg; joints [-0.165, -68.165, 222.083, -179.767, 24.281, -149.361]
  MoveL 47 to (14.22, -33.14, 34.03) mm, rotated rx 156.77 ry 6.58 rz 66.12 deg; joints [-0.029, -68.268, 222.31, -179.241, 24.448, -149.869]
  MoveL 48 to (14.26, -33.02, 34.01) mm, rotated rx 156.83 ry 6.63 rz 66.12 deg; joints [0.03, -68.286, 222.363, -179, 24.508, -150.105]
  MoveL 49 to (14.42, -32.61, 33.95) mm, rotated rx 156.96 ry 6.71 rz 66.13 deg; joints [0.148, -68.345, 222.483, -178.548, 24.594, -150.546]
  MoveL 50 to (14.83, -31.84, 33.87) mm, rotated rx 157.07 ry 6.83 rz 66.12 deg; joints [0.318, -68.457, 222.73, -177.976, 24.795, -151.06]
  MoveL 51 to (15.07, -31.48, 33.85) mm, rotated rx 157.23 ry 6.99 rz 66.11 deg; joints [0.502, -68.511, 222.905, -177.291, 25.015, -151.702]
  MoveL 52 to (15.75, -30.69, 33.86) mm, rotated rx 157.57 ry 7.32 rz 66.1 deg; joints [0.92, -68.634, 223.259, -175.814, 25.441, -153.077]
  MoveL 53 to (16.59, -29.95, 33.92) mm, rotated rx 157.95 ry 7.77 rz 66.07 deg; joints [1.43, -68.74, 223.679, -174.1, 26.059, -154.636]
  MoveL 54 to (16.71, -29.86, 33.93) mm, rotated rx 158.5 ry 8.24 rz 66.08 deg; joints [1.921, -68.731, 223.9, -172.259, 26.581, -156.45]
  MoveL 55 to (17.84, -29.15, 34.05) mm, rotated rx 159.6 ry 9.12 rz 66.14 deg; joints [3.014, -68.775, 224.362, -168.609, 27.583, -159.965]
  MoveL 56 to (19.12, -28.57, 34.21) mm, rotated rx 160.88 ry 10.22 rz 66.22 deg; joints [4.312, -68.705, 224.875, -164.643, 29.017, -163.745]
  MoveL 57 to (19.75, -28.34, 34.29) mm, rotated rx 162.15 ry 11.21 rz 66.36 deg; joints [5.439, -68.521, 225.187, -161.312, 30.319, -167.01]
  MoveL 58 to (21.31, -27.94, 34.48) mm, rotated rx 163.87 ry 12.43 rz 66.62 deg; joints [7.004, -68.226, 225.456, -157.113, 31.956, -171.081]
  MoveL 59 to (22.95, -27.7, 34.67) mm, rotated rx 171.55 ry 17.71 rz 87.41 deg; joints [-1.091, -67.529, 229.093, -188.447, 38.969, -167.256]
  MoveL 60 to (24.46, -27.64, 34.84) mm, rotated rx 173.85 ry 18.09 rz 88.09 deg; joints [0.48, -67.658, 229.368, -184.372, 39.128, -171.433]
  MoveL 61 to (26.05, -27.74, 35) mm, rotated rx 174.91 ry 18.23 rz 88.41 deg; joints [1.34, -67.69, 229.421, -182.34, 39.172, -173.396]
  Set speed (1000.0 mm/s)
  MoveL 62 to (26.05, -27.74, 35) mm, rotated rx 174.91 ry 18.23 rz 88.41 deg; joints [1.34, -67.69, 229.421, -182.34, 39.172, -173.396]
  MoveL 63 to (18.05, 3.66, 129.61) mm, rotated rx 174.91 ry 18.23 rz 88.41 deg; joints [0.057, -90.696, 232.799, -187.628, 19.656, -168.714]

--- program Path5 (robot Adept Viper s650) ---
  Smooth(1)
  Set speed (1000.0 mm/s)
  Set Ref.: Deburring Frame
  Set Tool: Spindle
  Show Spindle
  MoveJ 1 to (35.91, 14.91, 124.99) mm, rotated rx 179.25 ry 17.45 rz 89.78 deg; joints [6.005, -92.08, 234.127, -165.659, 18.922, 170.326]
  MoveL 2 to (35.91, 14.91, 124.99) mm, rotated rx 179.25 ry 17.45 rz 89.78 deg; joints [6.005, -92.08, 234.127, -165.659, 18.922, 170.326]
  MoveL 3 to (37.1, -15.07, 29.6) mm, rotated rx 179.25 ry 17.45 rz 89.78 deg; joints [5.683, -68.689, 231.217, -173.105, 39.071, 178.38]
  MoveL 4 to (37.1, -15.07, 29.6) mm, rotated rx 179.25 ry 17.45 rz 89.78 deg; joints [5.683, -68.689, 231.217, -173.105, 39.071, 178.38]
  Set speed (50.0 mm/s)
  MoveL 5 to (36.01, -14.68, 29.46) mm, rotated rx 179.59 ry 17.37 rz 89.88 deg; joints [5.707, -68.75, 231.239, -172.778, 38.966, 177.864]
  MoveL 6 to (34.84, -14.67, 29.46) mm, rotated rx -179.54 ry 17.36 rz 90.14 deg; joints [6.026, -68.725, 231.191, -171.619, 38.97, 176.445]
  MoveL 7 to (33.66, -14.8, 29.51) mm, rotated rx -178.68 ry 17.62 rz 90.4 deg; joints [6.345, -68.565, 231.328, -170.577, 39.567, 175.164]
  MoveL 8 to (32.57, -15.09, 29.62) mm, rotated rx -178 ry 17.96 rz 90.62 deg; joints [6.569, -68.351, 231.522, -169.874, 40.364, 174.254]
  MoveL 9 to (31.72, -15.42, 29.76) mm, rotated rx -177.42 ry 18.46 rz 90.82 deg; joints [6.775, -68.051, 231.826, -169.369, 41.507, 173.596]
  MoveL 10 to (30.83, -15.92, 29.97) mm, rotated rx -176.9 ry 19.05 rz 91.01 deg; joints [6.93, -67.687, 232.159, -169.038, 42.817, 173.112]
  MoveL 11 to (30.21, -16.39, 30.16) mm, rotated rx -176.52 ry 19.8 rz 91.18 deg; joints [7.042, -67.222, 232.613, -168.961, 44.498, 172.947]
  MoveL 12 to (29.59, -17.03, 30.43) mm, rotated rx -176.27 ry 20.59 rz 91.31 deg; joints [7.073, -66.704, 233.052, -169.087, 46.245, 172.993]
  MoveL 13 to (29.14, -17.68, 30.7) mm, rotated rx -176.25 ry 21.31 rz 91.37 deg; joints [7.004, -66.22, 233.429, -169.429, 47.807, 173.302]
  MoveL 14 to (28.81, -18.37, 30.99) mm, rotated rx -176.13 ry 21.98 rz 91.45 deg; joints [6.999, -65.733, 233.731, -169.608, 49.256, 173.447]
  MoveL 15 to (28.78, -18.46, 31.03) mm, rotated rx -176.3 ry 22.69 rz 91.43 deg; joints [6.907, -65.238, 234.176, -170.058, 50.866, 173.969]
  MoveL 16 to (28.6, -19.15, 31.33) mm, rotated rx -176.34 ry 23.16 rz 91.44 deg; joints [6.841, -64.866, 234.334, -170.3, 51.86, 174.208]
  MoveL 17 to (28.55, -19.86, 31.64) mm, rotated rx -176.46 ry 23.81 rz 91.43 deg; joints [6.763, -64.354, 234.576, -170.631, 53.236, 174.577]
  MoveL 18 to (28.57, -20.11, 31.75) mm, rotated rx -176.69 ry 24.36 rz 91.37 deg; joints [6.643, -63.914, 234.852, -171.036, 54.477, 175.06]
  MoveL 19 to (28.68, -20.81, 32.06) mm, rotated rx -176.83 ry 24.78 rz 91.33 deg; joints [6.583, -63.565, 234.939, -171.266, 55.312, 175.343]
  MoveL 20 to (28.93, -21.51, 32.37) mm, rotated rx -177.05 ry 25.23 rz 91.26 deg; joints [6.511, -63.183, 235.038, -171.541, 56.221, 175.708]
  MoveL 21 to (29.11, -21.86, 32.53) mm, rotated rx -177.27 ry 25.57 rz 91.18 deg; joints [6.431, -62.891, 235.149, -171.803, 56.949, 176.055]
  MoveL 22 to (29.55, -22.51, 32.82) mm, rotated rx -177.44 ry 25.79 rz 91.12 deg; joints [6.417, -62.695, 235.126, -171.931, 57.336, 176.28]
  MoveL 23 to (30.12, -23.12, 33.1) mm, rotated rx -177.65 ry 26.02 rz 91.03 deg; joints [6.409, -62.492, 235.112, -172.07, 57.741, 176.548]
  MoveL 24 to (30.22, -23.21, 33.14) mm, rotated rx -177.93 ry 26.18 rz 90.91 deg; joints [6.293, -62.365, 235.183, -172.35, 58.082, 176.907]
  MoveL 25 to (30.97, -23.77, 33.39) mm, rotated rx -178.21 ry 26.27 rz 90.79 deg; joints [6.284, -62.287, 235.112, -172.489, 58.171, 177.204]
  MoveL 26 to (31.84, -24.24, 33.6) mm, rotated rx -178.59 ry 26.39 rz 90.63 deg; joints [6.253, -62.184, 235.076, -172.701, 58.348, 177.621]
  MoveL 27 to (32.31, -24.44, 33.69) mm, rotated rx -179.02 ry 26.42 rz 90.44 deg; joints [6.134, -62.171, 235.066, -173.016, 58.372, 178.086]
  MoveL 28 to (33.36, -24.75, 33.83) mm, rotated rx -179.33 ry 26.44 rz 90.3 deg; joints [6.17, -62.15, 235.007, -173.111, 58.353, 178.396]
  MoveL 29 to (34.47, -24.93, 33.9) mm, rotated rx -179.69 ry 26.46 rz 90.14 deg; joints [6.189, -62.136, 234.976, -173.251, 58.348, 178.777]
  MoveL 30 to (34.64, -24.95, 33.91) mm, rotated rx 179.94 ry 26.44 rz 89.97 deg; joints [6.049, -62.169, 234.98, -173.557, 58.29, 179.171]
  MoveL 31 to (35.8, -24.96, 33.91) mm, rotated rx 179.59 ry 26.42 rz 89.82 deg; joints [6.087, -62.176, 234.967, -173.669, 58.258, 179.533]
  MoveL 32 to (36.96, -24.82, 33.85) mm, rotated rx 179.13 ry 26.38 rz 89.62 deg; joints [6.076, -62.216, 234.976, -173.878, 58.182, 180.007]
  MoveL 33 to (37.96, -24.56, 33.74) mm, rotated rx 178.71 ry 26.32 rz 89.43 deg; joints [6.054, -62.266, 235.005, -174.088, 58.105, 180.453]
  MoveL 34 to (38.96, -24.16, 33.56) mm, rotated rx 178.33 ry 26.23 rz 89.26 deg; joints [6.052, -62.345, 235.045, -174.255, 57.978, 180.843]
  MoveL 35 to (39.7, -23.73, 33.37) mm, rotated rx 178.02 ry 26.08 rz 89.13 deg; joints [6.029, -62.469, 235.068, -174.418, 57.743, 181.172]
  MoveL 36 to (40.46, -23.15, 33.11) mm, rotated rx 177.77 ry 25.87 rz 89.03 deg; joints [6.037, -62.655, 235.086, -174.516, 57.37, 181.417]
  MoveL 37 to (41.01, -22.58, 32.85) mm, rotated rx 177.57 ry 25.55 rz 88.95 deg; joints [6.017, -62.942, 235.049, -174.624, 56.733, 181.611]
  MoveL 38 to (41.49, -21.9, 32.54) mm, rotated rx 177.4 ry 25.12 rz 88.89 deg; joints [5.985, -63.322, 234.976, -174.731, 55.857, 181.769]
  MoveL 39 to (41.82, -21.19, 32.22) mm, rotated rx 177.26 ry 24.73 rz 88.85 deg; joints [5.947, -63.67, 234.919, -174.834, 55.061, 181.9]
  MoveL 40 to (42.01, -20.47, 31.9) mm, rotated rx 177.17 ry 24.42 rz 88.83 deg; joints [5.915, -63.939, 234.906, -174.911, 54.475, 181.989]
  MoveL 41 to (42.02, -20.38, 31.86) mm, rotated rx 177.1 ry 24.06 rz 88.82 deg; joints [5.847, -64.242, 234.735, -175.011, 53.645, 182.045]
  MoveL 42 to (42.03, -20.34, 31.84) mm, rotated rx 177.03 ry 23.66 rz 88.81 deg; joints [5.772, -64.571, 234.523, -175.117, 52.706, 182.099]
  MoveL 43 to (42.06, -19.64, 31.53) mm, rotated rx 176.95 ry 23.19 rz 88.8 deg; joints [5.695, -64.953, 234.405, -175.243, 51.742, 182.186]
  MoveL 44 to (41.97, -18.93, 31.22) mm, rotated rx 176.92 ry 22.55 rz 88.82 deg; joints [5.607, -65.462, 234.171, -175.35, 50.359, 182.199]
  MoveL 45 to (41.9, -18.65, 31.1) mm, rotated rx 176.86 ry 21.86 rz 88.83 deg; joints [5.49, -65.973, 233.797, -175.506, 48.786, 182.255]
  MoveL 46 to (41.64, -17.98, 30.82) mm, rotated rx 176.82 ry 21.31 rz 88.84 deg; joints [5.376, -66.378, 233.586, -175.657, 47.62, 182.305]
  MoveL 47 to (41.26, -17.33, 30.55) mm, rotated rx 176.93 ry 20.73 rz 88.91 deg; joints [5.316, -66.79, 233.328, -175.652, 46.365, 182.157]
  MoveL 48 to (41.19, -17.24, 30.51) mm, rotated rx 176.95 ry 20.07 rz 88.95 deg; joints [5.251, -67.204, 232.878, -175.692, 44.843, 182.095]
  MoveL 49 to (40.65, -16.62, 30.25) mm, rotated rx 177.17 ry 19.57 rz 89.05 deg; joints [5.238, -67.528, 232.645, -175.546, 43.786, 181.789]
  MoveL 50 to (39.98, -16.06, 30.02) mm, rotated rx 177.46 ry 18.95 rz 89.17 deg; joints [5.238, -67.91, 232.285, -175.302, 42.411, 181.343]
  MoveL 51 to (39.42, -15.7, 29.88) mm, rotated rx 177.87 ry 18.38 rz 89.33 deg; joints [5.333, -68.225, 231.898, -174.821, 41.136, 180.671]
  MoveL 52 to (38.51, -15.26, 29.69) mm, rotated rx 178.29 ry 17.98 rz 89.47 deg; joints [5.394, -68.446, 231.667, -174.372, 40.288, 180.007]
  MoveL 53 to (37.5, -14.93, 29.56) mm, rotated rx 178.38 ry 17.88 rz 89.5 deg; joints [5.277, -68.527, 231.667, -174.441, 40.097, 179.92]
  MoveL 54 to (37.15, -14.85, 29.53) mm, rotated rx 178.8 ry 17.59 rz 89.64 deg; joints [5.441, -68.66, 231.42, -173.839, 39.431, 179.191]
  Set speed (1000.0 mm/s)
  MoveL 55 to (37.15, -14.85, 29.53) mm, rotated rx 178.8 ry 17.59 rz 89.64 deg; joints [5.441, -68.66, 231.42, -173.839, 39.431, 179.191]
  MoveL 56 to (35.24, 15.37, 124.83) mm, rotated rx 178.8 ry 17.59 rz 89.64 deg; joints [5.615, -92.216, 234.449, -167.555, 19.152, 172.278]

--- program Path6 (robot Adept Viper s650) ---
  Smooth(1)
  Set speed (1000.0 mm/s)
  Set Ref.: Deburring Frame
  Set Tool: Spindle
  Show Spindle
  MoveJ 1 to (15.93, 14.63, 123.58) mm, rotated rx 174.49 ry 8.02 rz 89.23 deg; joints [-1.343, -88.996, 222.846, 101.575, 4.795, -98.532]
  MoveL 2 to (15.93, 14.63, 123.58) mm, rotated rx 174.49 ry 8.02 rz 89.23 deg; joints [-1.343, -88.996, 222.846, 101.575, 4.795, -98.532]
  MoveL 3 to (25.34, 0.63, 25.01) mm, rotated rx 174.49 ry 8.02 rz 89.23 deg; joints [0.17, -72.134, 225.959, 170.082, 21.305, -166.634]
  MoveL 4 to (25.34, 0.63, 25.01) mm, rotated rx 174.49 ry 8.02 rz 89.23 deg; joints [0.17, -72.134, 225.959, 170.082, 21.305, -166.634]
  Set speed (50.0 mm/s)
  MoveL 5 to (24.79, 0.21, 25.02) mm, rotated rx 174.25 ry 7.62 rz 89.24 deg; joints [-0.107, -72.028, 225.415, 168.579, 20.551, -165.212]
  MoveL 6 to (23.87, -0.3, 24.99) mm, rotated rx 172.74 ry 8.2 rz 88.96 deg; joints [-1.232, -71.82, 225.987, 164.621, 22.304, -161.269]
  MoveL 7 to (23.04, -0.63, 24.92) mm, rotated rx 170.31 ry 9.91 rz 88.32 deg; joints [-2.836, -71.385, 227.804, 161.174, 26.874, -157.714]
  MoveL 8 to (21.91, -0.94, 24.77) mm, rotated rx 168.13 ry 10.71 rz 87.76 deg; joints [-4.355, -70.81, 228.557, 157.731, 29.701, -154.264]
  MoveL 9 to (20.75, -1.11, 24.54) mm, rotated rx 166.03 ry 10.84 rz 87.32 deg; joints [-5.872, -70.206, 228.576, 153.78, 31.314, -150.362]
  MoveL 10 to (19.51, -1.15, 24.22) mm, rotated rx 163.87 ry 10.92 rz 86.86 deg; joints [-7.422, -69.49, 228.528, 150.064, 33.04, -146.711]
  MoveL 11 to (18.29, -1.04, 23.82) mm, rotated rx 162.13 ry 10.8 rz 86.54 deg; joints [-8.705, -68.853, 228.286, 146.955, 34.218, -143.709]
  MoveL 12 to (18.07, -1.01, 23.74) mm, rotated rx 160.85 ry 10.34 rz 86.43 deg; joints [-9.59, -68.427, 227.692, 144.02, 34.443, -140.782]
  MoveL 13 to (16.93, -0.73, 23.29) mm, rotated rx 159.49 ry 10.29 rz 86.18 deg; joints [-10.602, -67.832, 227.544, 141.949, 35.601, -138.83]
  MoveL 14 to (15.89, -0.32, 22.8) mm, rotated rx 158.36 ry 10.34 rz 85.93 deg; joints [-11.442, -67.299, 227.54, 140.556, 36.768, -137.555]
  MoveL 15 to (15.39, -0.06, 22.55) mm, rotated rx 157.52 ry 9.55 rz 86.07 deg; joints [-12.14, -66.971, 226.592, 137.502, 36.282, -134.608]
  MoveL 16 to (14.61, 0.48, 22.13) mm, rotated rx 157.08 ry 8.92 rz 86.25 deg; joints [-12.622, -66.772, 225.886, 135.234, 35.806, -132.505]
  MoveL 17 to (13.95, 1.14, 21.73) mm, rotated rx 157.14 ry 8.66 rz 86.37 deg; joints [-12.745, -66.797, 225.709, 134.551, 35.487, -131.971]
  MoveL 18 to (13.53, 1.71, 21.46) mm, rotated rx 157.45 ry 8.31 rz 86.57 deg; joints [-12.688, -66.951, 225.435, 133.883, 34.764, -131.425]
  MoveL 19 to (13.21, 2.37, 21.21) mm, rotated rx 158.34 ry 8.06 rz 86.81 deg; joints [-12.252, -67.377, 225.389, 134.218, 33.672, -131.882]
  MoveL 20 to (13.03, 2.93, 21.06) mm, rotated rx 160.75 ry 7.98 rz 87.23 deg; joints [-10.825, -68.407, 225.69, 137.096, 31.452, -134.885]
  MoveL 21 to (12.95, 3.5, 20.94) mm, rotated rx 160.34 ry 7.16 rz 87.45 deg; joints [-11.194, -68.27, 224.797, 134.115, 30.656, -131.969]
  MoveL 22 to (12.93, 3.77, 20.9) mm, rotated rx 157.6 ry 6.14 rz 87.48 deg; joints [-12.988, -67.052, 223.235, 127.511, 31.867, -125.359]
  MoveL 23 to (12.94, 4.05, 20.87) mm, rotated rx 156.92 ry 5.77 rz 87.55 deg; joints [-13.444, -66.729, 222.726, 125.587, 32.099, -123.449]
  MoveL 24 to (12.97, 4.32, 20.85) mm, rotated rx 157.1 ry 5.41 rz 87.72 deg; joints [-13.369, -66.796, 222.359, 124.602, 31.51, -122.494]
  MoveL 25 to (13.04, 4.68, 20.84) mm, rotated rx 158.83 ry 4.68 rz 88.19 deg; joints [-12.362, -67.489, 221.77, 123.96, 28.956, -121.927]
  MoveL 26 to (13.11, 4.97, 20.85) mm, rotated rx 159.54 ry 4.02 rz 88.5 deg; joints [-11.957, -67.698, 221.089, 122.352, 27.519, -120.359]
  MoveL 27 to (13.21, 5.25, 20.86) mm, rotated rx 158.15 ry 3.75 rz 88.5 deg; joints [-12.843, -67.083, 220.574, 119.805, 28.678, -117.796]
  MoveL 28 to (13.47, 5.79, 20.93) mm, rotated rx 157.06 ry 3.41 rz 88.56 deg; joints [-13.513, -66.612, 220.078, 117.558, 29.494, -115.534]
  MoveL 29 to (13.67, 6.1, 21) mm, rotated rx 156.35 ry 3.03 rz 88.68 deg; joints [-13.953, -66.24, 219.507, 115.517, 29.898, -113.484]
  MoveL 30 to (14.15, 6.68, 21.17) mm, rotated rx 155.9 ry 2.57 rz 88.85 deg; joints [-14.201, -66.031, 218.948, 113.492, 29.978, -111.434]
  MoveL 31 to (14.42, 6.95, 21.28) mm, rotated rx 155.69 ry 2.05 rz 89.07 deg; joints [-14.327, -65.835, 218.268, 111.399, 29.813, -109.333]
  MoveL 32 to (15.18, 7.53, 21.61) mm, rotated rx 156.07 ry 0.82 rz 89.64 deg; joints [-14.05, -65.76, 216.762, 106.796, 28.554, -104.702]
  MoveL 33 to (16.1, 8.02, 22.01) mm, rotated rx 156.55 ry -0.17 rz 90.07 deg; joints [-13.663, -65.776, 215.597, 103.011, 27.462, -100.856]
  MoveL 34 to (16.22, 8.08, 22.06) mm, rotated rx 156.87 ry -0.13 rz 90.05 deg; joints [-13.453, -65.966, 215.748, 103.376, 27.12, -101.21]
  MoveL 35 to (17.38, 8.47, 22.55) mm, rotated rx 158.13 ry -0.41 rz 90.16 deg; joints [-12.522, -66.609, 215.734, 102.85, 25.482, -100.576]
  MoveL 36 to (18.62, 8.71, 23.02) mm, rotated rx 159.98 ry -0.93 rz 90.34 deg; joints [-11.187, -67.327, 215.427, 101.373, 23.061, -98.986]
  MoveL 37 to (19.26, 8.77, 23.25) mm, rotated rx 161.74 ry 0.59 rz 89.81 deg; joints [-9.92, -68.706, 217.884, 110.354, 21.758, -107.856]
  MoveL 38 to (20.49, 8.77, 23.63) mm, rotated rx 163.91 ry 0.71 rz 89.79 deg; joints [-8.301, -69.595, 218.358, 113.447, 19.293, -110.813]
  MoveL 39 to (21.7, 8.64, 23.95) mm, rotated rx 166.25 ry -1.22 rz 90.3 deg; joints [-6.598, -69.538, 215.92, 103.8, 15.346, -101.108]
  MoveL 40 to (22.56, 8.45, 24.14) mm, rotated rx 168.76 ry -0.27 rz 90.05 deg; joints [-4.718, -70.563, 217.389, 114.542, 12.893, -111.743]
  MoveL 41 to (23.61, 8.1, 24.33) mm, rotated rx 171.04 ry 0.23 rz 89.96 deg; joints [-2.954, -71.164, 218.09, 124.864, 10.748, -121.951]
  MoveL 42 to (24.57, 7.63, 24.46) mm, rotated rx 172.3 ry -0.67 rz 90.09 deg; joints [-1.966, -70.914, 216.786, 120.305, 8.416, -117.332]
  MoveL 43 to (24.7, 7.56, 24.47) mm, rotated rx 172.94 ry -0.86 rz 90.11 deg; joints [-1.499, -70.896, 216.514, 120.54, 7.521, -117.57]
  MoveL 44 to (25.41, 7.04, 24.55) mm, rotated rx 175.32 ry 1.1 rz 89.91 deg; joints [0.368, -71.791, 218.987, 155.677, 8.126, -152.596]
  MoveL 45 to (25.99, 6.47, 24.61) mm, rotated rx 177.48 ry 2.89 rz 89.87 deg; joints [2.066, -72.326, 221.059, 177.359, 10.692, -174.188]
  MoveL 46 to (26.06, 6.39, 24.61) mm, rotated rx 177.49 ry 2.59 rz 89.89 deg; joints [2.064, -72.227, 220.661, 177.115, 10.096, -173.951]
  MoveL 47 to (26.46, 5.81, 24.66) mm, rotated rx 177.43 ry 2.61 rz 89.88 deg; joints [2.078, -72.138, 220.554, 176.918, 10.107, -173.704]
  MoveL 48 to (26.75, 5.21, 24.7) mm, rotated rx 177.77 ry 2.9 rz 89.89 deg; joints [2.374, -72.12, 220.751, 179.613, 10.578, -176.366]
  MoveL 49 to (26.78, 5.12, 24.7) mm, rotated rx 177.72 ry 3.22 rz 89.87 deg; joints [2.357, -72.193, 221.135, 179.469, 11.21, -176.201]
  MoveL 50 to (26.94, 4.51, 24.74) mm, rotated rx 178.07 ry 3.6 rz 89.88 deg; joints [2.649, -72.19, 221.452, 181.842, 11.906, -178.552]
  MoveL 51 to (27, 3.91, 24.78) mm, rotated rx 178.08 ry 3.88 rz 89.87 deg; joints [2.672, -72.16, 221.654, 181.934, 12.417, -178.628]
  MoveL 52 to (27, 3.9, 24.78) mm, rotated rx 178.1 ry 4.2 rz 89.86 deg; joints [2.701, -72.234, 222.051, 182.067, 13.062, -178.747]
  MoveL 53 to (27, 3.7, 24.8) mm, rotated rx 178.08 ry 4.44 rz 89.85 deg; joints [2.697, -72.255, 222.299, 181.984, 13.531, -178.653]
  MoveL 54 to (26.91, 3.07, 24.84) mm, rotated rx 178.1 ry 4.74 rz 89.84 deg; joints [2.71, -72.216, 222.513, 182.081, 14.08, -178.751]
  MoveL 55 to (26.82, 2.74, 24.87) mm, rotated rx 177.4 ry 5.41 rz 89.75 deg; joints [2.245, -72.292, 223.286, 178.969, 15.472, -175.592]
  MoveL 56 to (26.7, 2.41, 24.89) mm, rotated rx 178.08 ry 5.06 rz 89.83 deg; joints [2.68, -72.175, 222.748, 181.946, 14.674, -178.629]
  MoveL 57 to (26.36, 1.77, 24.94) mm, rotated rx 176.73 ry 5.99 rz 89.66 deg; joints [1.735, -72.225, 223.789, 176.256, 16.68, -172.882]
  Set speed (1000.0 mm/s)
  MoveL 58 to (26.36, 1.77, 24.94) mm, rotated rx 176.73 ry 5.99 rz 89.66 deg; joints [1.735, -72.225, 223.789, 176.256, 16.68, -172.882]
  MoveL 59 to (20.71, 12.22, 124.23) mm, rotated rx 178.98 ry 6.75 rz 109.77 deg; joints [-8.858, -84.012, 216.145, 74.27, 21.663, -93.453]

--- program Path7 (robot Adept Viper s650) ---
  Smooth(1)
  Set speed (1000.0 mm/s)
  Set Ref.: Deburring Frame
  Set Tool: Spindle
  Show Spindle
  MoveJ 1 to (69.75, 0.94, 121.32) mm, rotated rx -167.39 ry -4.29 rz 89.04 deg; joints [17.431, -72.726, 197.168, -41.431, 31.022, 44.967]
  MoveL 2 to (69.75, 0.94, 121.32) mm, rotated rx -167.39 ry -4.29 rz 89.04 deg; joints [17.431, -72.726, 197.168, -41.431, 31.022, 44.967]
  MoveL 3 to (48.06, 8.6, 24.01) mm, rotated rx -167.39 ry -4.29 rz 89.04 deg; joints [15.011, -66.036, 208.443, -73.936, 19.458, 78.7]
  MoveL 4 to (48.06, 8.6, 24.01) mm, rotated rx -167.39 ry -4.29 rz 89.04 deg; joints [15.011, -66.036, 208.443, -73.936, 19.458, 78.7]
  Set speed (50.0 mm/s)
  MoveL 5 to (46.89, 8.29, 24.24) mm, rotated rx -168.06 ry -4.06 rz 89.14 deg; joints [14.446, -66.446, 208.971, -74.878, 18.512, 79.552]
  MoveL 6 to (46.77, 8.25, 24.26) mm, rotated rx -169.17 ry -3.92 rz 89.25 deg; joints [13.724, -66.913, 209.478, -75.181, 17.162, 79.903]
  MoveL 7 to (45.77, 7.82, 24.42) mm, rotated rx -170.36 ry -3.72 rz 89.37 deg; joints [12.822, -67.403, 210.037, -75.857, 15.623, 80.524]
  MoveL 8 to (44.9, 7.28, 24.52) mm, rotated rx -171.62 ry -2.94 rz 89.57 deg; joints [11.927, -68.146, 211.37, -80.981, 13.87, 85.637]
  MoveL 9 to (44.39, 6.86, 24.57) mm, rotated rx -172.35 ry -2.06 rz 89.72 deg; joints [11.434, -68.743, 212.709, -88.211, 12.911, 92.882]
  MoveL 10 to (43.83, 6.25, 24.63) mm, rotated rx -172.8 ry -1.04 rz 89.87 deg; joints [11.123, -69.255, 214.095, -97.197, 12.549, 101.866]
  MoveL 11 to (43.48, 5.7, 24.66) mm, rotated rx -173.14 ry 0.16 rz 90.02 deg; joints [10.928, -69.77, 215.682, -107.761, 12.782, 112.461]
  MoveL 12 to (43.2, 5.07, 24.71) mm, rotated rx -173.42 ry 1.19 rz 90.14 deg; joints [10.76, -70.138, 216.977, -116.31, 13.316, 121.036]
  MoveL 13 to (43.16, 4.96, 24.71) mm, rotated rx -173.54 ry 1.97 rz 90.22 deg; joints [10.728, -70.417, 218.002, -122.038, 14.029, 126.81]
  MoveL 14 to (43.03, 4.35, 24.75) mm, rotated rx -173.56 ry 2.91 rz 90.33 deg; joints [10.743, -70.619, 219.08, -127.719, 15.125, 132.52]
  MoveL 15 to (43, 3.84, 24.79) mm, rotated rx -173.7 ry 3.82 rz 90.42 deg; joints [10.698, -70.815, 220.14, -132.821, 16.244, 137.67]
  MoveL 16 to (43, 3.72, 24.8) mm, rotated rx -173.75 ry 4.36 rz 90.48 deg; joints [10.693, -70.934, 220.79, -135.456, 16.989, 140.341]
  MoveL 17 to (43.03, 3.43, 24.82) mm, rotated rx -173.79 ry 5.02 rz 90.55 deg; joints [10.706, -71.035, 221.545, -138.304, 17.977, 143.23]
  MoveL 18 to (43.16, 2.82, 24.86) mm, rotated rx -173.86 ry 6.06 rz 90.65 deg; joints [10.726, -71.128, 222.657, -142.167, 19.587, 147.168]
  MoveL 19 to (43.39, 2.21, 24.91) mm, rotated rx -173.81 ry 7 rz 90.76 deg; joints [10.83, -71.135, 223.608, -144.839, 21.193, 149.917]
  MoveL 20 to (43.44, 2.11, 24.92) mm, rotated rx -173.8 ry 7.61 rz 90.82 deg; joints [10.878, -71.17, 224.297, -146.486, 22.286, 151.613]
  MoveL 21 to (43.82, 1.51, 24.96) mm, rotated rx -173.77 ry 8.34 rz 90.91 deg; joints [10.979, -71.1, 224.973, -148.102, 23.6, 153.313]
  MoveL 22 to (44.33, 0.93, 25) mm, rotated rx -173.43 ry 9.23 rz 91.06 deg; joints [11.31, -70.932, 225.759, -149.113, 25.395, 154.419]
  MoveL 23 to (44.7, 0.59, 25.01) mm, rotated rx -172.98 ry 9.9 rz 91.21 deg; joints [11.678, -70.75, 226.319, -149.366, 26.843, 154.736]
  MoveL 24 to (45.11, 0.29, 25.02) mm, rotated rx -172.46 ry 10.32 rz 91.36 deg; joints [12.083, -70.543, 226.603, -148.971, 27.886, 154.382]
  MoveL 25 to (45.95, -0.21, 24.99) mm, rotated rx -171.48 ry 10.85 rz 91.62 deg; joints [12.84, -70.145, 226.852, -147.794, 29.372, 153.273]
  MoveL 26 to (46.71, -0.54, 24.94) mm, rotated rx -170.03 ry 11.41 rz 91.99 deg; joints [13.865, -69.602, 227.074, -145.983, 31.187, 151.49]
  MoveL 27 to (47.79, -0.88, 24.81) mm, rotated rx -168.29 ry 11.9 rz 92.45 deg; joints [15.097, -68.891, 227.125, -143.712, 33.094, 149.253]
  MoveL 28 to (48.93, -1.08, 24.61) mm, rotated rx -166.6 ry 12.44 rz 92.94 deg; joints [16.274, -68.125, 227.253, -141.968, 35.137, 147.559]
  MoveL 29 to (49.45, -1.13, 24.49) mm, rotated rx -165.18 ry 12.74 rz 93.34 deg; joints [17.18, -67.508, 227.227, -140.44, 36.574, 146.002]
  MoveL 30 to (50.67, -1.14, 24.17) mm, rotated rx -163.52 ry 12.89 rz 93.78 deg; joints [18.308, -66.714, 226.956, -138.364, 38, 143.953]
  MoveL 31 to (51.88, -1.01, 23.76) mm, rotated rx -161.93 ry 13.03 rz 94.21 deg; joints [19.379, -65.908, 226.705, -136.552, 39.422, 142.178]
  MoveL 32 to (52.36, -0.92, 23.58) mm, rotated rx -160.76 ry 13.06 rz 94.51 deg; joints [20.095, -65.342, 226.46, -135.22, 40.339, 140.805]
  MoveL 33 to (53.49, -0.59, 23.1) mm, rotated rx -159.74 ry 12.95 rz 94.73 deg; joints [20.827, -64.793, 226.096, -133.751, 40.999, 139.404]
  MoveL 34 to (54.5, -0.12, 22.61) mm, rotated rx -159.13 ry 12.65 rz 94.77 deg; joints [21.339, -64.468, 225.647, -132.331, 41.084, 138.069]
  MoveL 35 to (54.6, -0.07, 22.56) mm, rotated rx -159.05 ry 12.42 rz 94.71 deg; joints [21.405, -64.461, 225.379, -131.717, 40.784, 137.441]
  MoveL 36 to (55.4, 0.49, 22.12) mm, rotated rx -159.32 ry 12.06 rz 94.51 deg; joints [21.416, -64.587, 225.11, -131.1, 40.136, 136.971]
  MoveL 37 to (56.04, 1.13, 21.74) mm, rotated rx -159.77 ry 11.4 rz 94.17 deg; joints [21.312, -64.857, 224.573, -129.962, 38.882, 135.948]
  MoveL 38 to (56.38, 1.58, 21.52) mm, rotated rx -160.32 ry 10.65 rz 93.78 deg; joints [21.091, -65.178, 223.938, -128.692, 37.407, 134.735]
  MoveL 39 to (56.73, 2.21, 21.27) mm, rotated rx -160.83 ry 9.81 rz 93.39 deg; joints [20.883, -65.479, 223.214, -127.083, 35.861, 133.18]
  MoveL 40 to (56.88, 2.61, 21.14) mm, rotated rx -161.25 ry 8.88 rz 93 deg; joints [20.677, -65.695, 222.317, -125.041, 34.298, 131.131]
  MoveL 41 to (57.02, 3.19, 21) mm, rotated rx -161.52 ry 7.93 rz 92.64 deg; joints [20.547, -65.826, 221.372, -122.62, 32.889, 128.7]
  MoveL 42 to (57.05, 3.5, 20.94) mm, rotated rx -161.62 ry 7.16 rz 92.37 deg; joints [20.48, -65.837, 220.525, -120.394, 31.882, 126.433]
  MoveL 43 to (57.06, 3.71, 20.91) mm, rotated rx -161.66 ry 6.46 rz 92.14 deg; joints [20.437, -65.796, 219.722, -118.227, 31.06, 124.221]
  MoveL 44 to (57.05, 4.19, 20.86) mm, rotated rx -161.61 ry 5.61 rz 91.86 deg; joints [20.444, -65.7, 218.738, -115.343, 30.224, 121.285]
  MoveL 45 to (57.01, 4.46, 20.85) mm, rotated rx -161.47 ry 4.83 rz 91.62 deg; joints [20.489, -65.519, 217.757, -112.482, 29.614, 118.356]
  MoveL 46 to (56.95, 4.73, 20.84) mm, rotated rx -161.3 ry 4.17 rz 91.41 deg; joints [20.553, -65.328, 216.907, -109.938, 29.211, 115.752]
  MoveL 47 to (56.88, 5, 20.85) mm, rotated rx -161.11 ry 3.63 rz 91.24 deg; joints [20.63, -65.142, 216.195, -107.765, 28.972, 113.526]
  MoveL 48 to (56.85, 5.09, 20.85) mm, rotated rx -160.88 ry 3.03 rz 91.05 deg; joints [20.721, -64.875, 215.335, -105.288, 28.774, 110.983]
  MoveL 49 to (56.62, 5.62, 20.91) mm, rotated rx -160.37 ry 2.03 rz 90.72 deg; joints [20.932, -64.408, 213.938, -101.078, 28.693, 106.658]
  MoveL 50 to (56.29, 6.15, 21.01) mm, rotated rx -159.59 ry 0.86 rz 90.32 deg; joints [21.269, -63.692, 212.161, -96.043, 28.995, 101.464]
  MoveL 51 to (55.85, 6.68, 21.17) mm, rotated rx -158.73 ry -0.19 rz 89.92 deg; joints [21.626, -62.938, 210.483, -91.593, 29.596, 96.847]
  MoveL 52 to (55.27, 7.21, 21.41) mm, rotated rx -157.96 ry -1.1 rz 89.55 deg; joints [21.92, -62.255, 209.006, -87.903, 30.276, 92.991]
  MoveL 53 to (54.46, 7.74, 21.76) mm, rotated rx -157.55 ry -1.86 rz 89.23 deg; joints [21.993, -61.837, 207.89, -85.027, 30.658, 89.968]
  MoveL 54 to (53.52, 8.18, 22.17) mm, rotated rx -157.84 ry -2.47 rz 89 deg; joints [21.663, -61.872, 207.261, -82.847, 30.316, 87.688]
  MoveL 55 to (52.46, 8.51, 22.61) mm, rotated rx -158.65 ry -3.06 rz 88.8 deg; joints [21.016, -62.181, 206.845, -80.707, 29.428, 85.471]
  MoveL 56 to (52.24, 8.56, 22.7) mm, rotated rx -159.63 ry -3.36 rz 88.75 deg; joints [20.387, -62.583, 206.814, -79.57, 28.367, 84.366]
  MoveL 57 to (50.98, 8.75, 23.17) mm, rotated rx -161.22 ry -3.58 rz 88.78 deg; joints [19.284, -63.45, 207.237, -78.665, 26.548, 83.43]
  MoveL 58 to (49.69, 8.78, 23.58) mm, rotated rx -162.27 ry -3.83 rz 88.78 deg; joints [18.467, -63.963, 207.355, -77.539, 25.329, 82.22]
  Set speed (1000.0 mm/s)
  MoveL 59 to (49.69, 8.78, 23.58) mm, rotated rx -162.27 ry -3.83 rz 88.78 deg; joints [18.467, -63.963, 207.355, -77.539, 25.329, 82.22]
  MoveL 60 to (80, 1.77, 118.62) mm, rotated rx -162.27 ry -3.83 rz 88.78 deg; joints [21.783, -70.136, 195.909, -49.726, 35.58, 52.965]

--- program telephone (robot Adept Viper s650) ---
  Smooth(1)
  Set speed (1000.0 mm/s)
  Set Ref.: Deburring Frame
  Set Tool: Spindle
  Show Spindle
  MoveJ 1 to (12.14, -1.28, 123.53) mm, rotated rx 171.24 ry -25.98 rz 93.86 deg; joints [-3.536, -50.57, 156.892, 9.61, 61.633, -6.336]
  MoveL 2 to (12.14, -1.28, 123.53) mm, rotated rx 171.24 ry -25.98 rz 93.86 deg; joints [-3.536, -50.57, 156.892, 9.61, 61.633, -6.336]
  MoveL 3 to (24.42, 42.94, 34.69) mm, rotated rx 171.24 ry -25.98 rz 93.86 deg; joints [-2.466, -57.53, 184.325, 12.493, 41.346, -10.125]
  MoveL 4 to (24.42, 42.94, 34.69) mm, rotated rx 171.24 ry -25.98 rz 93.86 deg; joints [-2.466, -57.53, 184.325, 12.493, 41.346, -10.125]
  Set speed (50.0 mm/s)
  MoveL 5 to (22.55, 42.5, 34.21) mm, rotated rx 169.14 ry -25.98 rz 94.8 deg; joints [-3.898, -56.96, 183.877, 15.571, 42.025, -13.412]
  MoveL 6 to (20.76, 41.97, 33.57) mm, rotated rx 165.79 ry -25.76 rz 96.28 deg; joints [-6.039, -56.114, 183.403, 20.346, 43.079, -18.399]
  MoveL 7 to (20.38, 41.84, 33.41) mm, rotated rx 163.49 ry -25.66 rz 97.32 deg; joints [-7.383, -55.385, 182.881, 23.335, 44.116, -21.446]
  MoveL 8 to (18.76, 41.21, 32.62) mm, rotated rx 160.79 ry -25.62 rz 98.57 deg; joints [-9.025, -54.084, 181.775, 26.499, 45.7, -24.776]
  MoveL 9 to (17.27, 40.5, 31.73) mm, rotated rx 157.85 ry -25.29 rz 99.87 deg; joints [-10.781, -52.764, 180.885, 29.938, 47.243, -28.364]
  MoveL 10 to (15.95, 39.69, 30.78) mm, rotated rx 155.92 ry -24.87 rz 100.65 deg; joints [-11.971, -51.891, 180.467, 32.275, 48.105, -30.827]
  MoveL 11 to (15.41, 39.29, 30.34) mm, rotated rx 155.14 ry -24.61 rz 100.92 deg; joints [-12.466, -51.6, 180.444, 33.316, 48.347, -31.92]
  MoveL 12 to (14.51, 38.45, 29.5) mm, rotated rx 155.05 ry -24.44 rz 100.89 deg; joints [-12.625, -51.457, 180.456, 33.623, 48.209, -32.308]
  MoveL 13 to (13.81, 37.57, 28.74) mm, rotated rx 155.3 ry -24.25 rz 100.7 deg; joints [-12.596, -51.552, 180.708, 33.674, 47.757, -32.421]
  MoveL 14 to (13.7, 37.39, 28.6) mm, rotated rx 155.69 ry -24.05 rz 100.43 deg; joints [-12.456, -51.943, 181.26, 33.619, 47.169, -32.391]
  MoveL 15 to (13.29, 36.58, 28.01) mm, rotated rx 156.27 ry -23.67 rz 100.01 deg; joints [-12.266, -52.483, 182.106, 33.643, 46.162, -32.463]
  MoveL 16 to (13.05, 35.75, 27.49) mm, rotated rx 156.9 ry -23.16 rz 99.52 deg; joints [-12.054, -53.179, 183.199, 33.792, 44.946, -32.648]
  MoveL 17 to (13, 35.49, 27.35) mm, rotated rx 157.32 ry -22.64 rz 99.14 deg; joints [-11.935, -53.907, 184.349, 34.157, 43.873, -33.041]
  MoveL 18 to (12.96, 34.76, 26.99) mm, rotated rx 157.65 ry -21.99 rz 98.75 deg; joints [-11.88, -54.608, 185.575, 34.844, 42.695, -33.745]
  MoveL 19 to (12.99, 34.34, 26.8) mm, rotated rx 157.86 ry -21.19 rz 98.37 deg; joints [-11.9, -55.463, 187.084, 35.902, 41.406, -34.825]
  MoveL 20 to (13.12, 33.68, 26.56) mm, rotated rx 157.9 ry -20.36 rz 98.04 deg; joints [-12.003, -56.193, 188.494, 37.259, 40.236, -36.184]
  MoveL 21 to (13.22, 33.35, 26.46) mm, rotated rx 157.8 ry -19.62 rz 97.8 deg; joints [-12.169, -56.831, 189.765, 38.686, 39.301, -37.62]
  MoveL 22 to (13.39, 32.93, 26.36) mm, rotated rx 157.64 ry -18.96 rz 97.61 deg; joints [-12.347, -57.318, 190.808, 40.077, 38.564, -39.006]
  MoveL 23 to (13.54, 32.63, 26.3) mm, rotated rx 157.43 ry -18.36 rz 97.46 deg; joints [-12.544, -57.736, 191.744, 41.458, 37.964, -40.384]
  MoveL 24 to (13.72, 32.32, 26.25) mm, rotated rx 157.2 ry -17.83 rz 97.33 deg; joints [-12.737, -58.081, 192.56, 42.778, 37.474, -41.695]
  MoveL 25 to (13.92, 32.02, 26.22) mm, rotated rx 156.94 ry -17.29 rz 97.21 deg; joints [-12.946, -58.405, 193.36, 44.174, 37.03, -43.079]
  MoveL 26 to (14.19, 31.67, 26.21) mm, rotated rx 156.65 ry -16.75 rz 97.09 deg; joints [-13.16, -58.702, 194.137, 45.625, 36.628, -44.509]
  MoveL 27 to (14.48, 31.34, 26.21) mm, rotated rx 156.3 ry -16.15 rz 96.96 deg; joints [-13.413, -59.016, 194.987, 47.291, 36.236, -46.153]
  MoveL 28 to (15.2, 30.67, 26.29) mm, rotated rx 156.06 ry -15.56 rz 96.79 deg; joints [-13.543, -59.342, 195.805, 48.86, 35.761, -47.638]
  MoveL 29 to (15.39, 30.51, 26.32) mm, rotated rx 156 ry -15.2 rz 96.66 deg; joints [-13.609, -59.614, 196.386, 49.771, 35.41, -48.533]
  MoveL 30 to (16.45, 29.77, 26.54) mm, rotated rx 156.49 ry -15.03 rz 96.44 deg; joints [-13.207, -59.972, 196.75, 49.654, 34.722, -48.272]
  MoveL 31 to (17.69, 29.09, 26.83) mm, rotated rx 157.93 ry -14.89 rz 95.95 deg; joints [-12.223, -60.796, 197.412, 48.421, 33.184, -46.868]
  MoveL 32 to (18.56, 28.69, 27.03) mm, rotated rx 160.05 ry -15.06 rz 95.39 deg; joints [-10.811, -61.636, 197.763, 45.376, 31.433, -43.69]
  MoveL 33 to (20.41, 27.99, 27.42) mm, rotated rx 163.33 ry -15.42 rz 94.55 deg; joints [-8.509, -62.625, 197.94, 39.53, 29.1, -37.582]
  MoveL 34 to (22.41, 27.39, 27.74) mm, rotated rx 167.97 ry -15.69 rz 93.3 deg; joints [-5.265, -63.787, 198.29, 29.873, 26.188, -27.648]
  MoveL 35 to (24.72, 26.86, 27.96) mm, rotated rx 173.05 ry -15.74 rz 91.89 deg; joints [-1.62, -64.627, 198.589, 16.994, 23.849, -14.476]
  MoveL 36 to (26.94, 26.48, 28.02) mm, rotated rx 177.16 ry -15.47 rz 90.76 deg; joints [1.414, -65.073, 198.965, 5.062, 22.6, -2.286]
  MoveL 37 to (29.23, 26.19, 27.99) mm, rotated rx 179.49 ry -15.12 rz 90.13 deg; joints [3.274, -65.257, 199.299, -2.315, 22.108, 5.34]
  MoveL 38 to (31.61, 25.99, 27.93) mm, rotated rx -179.8 ry -14.85 rz 89.95 deg; joints [4.06, -65.378, 199.587, -4.948, 21.782, 8.225]
  MoveL 39 to (33.74, 25.91, 27.9) mm, rotated rx -179.92 ry -14.72 rz 89.98 deg; joints [4.25, -65.454, 199.754, -4.948, 21.558, 8.447]
  MoveL 40 to (36.85, 25.93, 27.91) mm, rotated rx 179.83 ry -14.7 rz 90.04 deg; joints [4.471, -65.451, 199.756, -4.618, 21.515, 8.439]
  MoveL 41 to (39.96, 26.13, 27.97) mm, rotated rx -179.74 ry -14.75 rz 89.93 deg; joints [5.142, -65.371, 199.612, -6.326, 21.73, 10.468]
  MoveL 42 to (43.06, 26.52, 28.03) mm, rotated rx -177.4 ry -14.79 rz 89.34 deg; joints [7.095, -65.047, 199.181, -13.559, 22.646, 18.013]
  MoveL 43 to (45.43, 26.95, 27.97) mm, rotated rx -173.92 ry -14.89 rz 88.43 deg; joints [9.687, -64.26, 198.3, -22.661, 24.653, 27.328]
  MoveL 44 to (46.34, 27.15, 27.91) mm, rotated rx -170.44 ry -14.73 rz 87.55 deg; joints [12.068, -63.373, 197.578, -30.431, 26.844, 35.146]
  MoveL 45 to (48.46, 27.71, 27.65) mm, rotated rx -166.38 ry -14.38 rz 86.55 deg; joints [14.925, -62.106, 196.758, -38.128, 29.784, 42.993]
  MoveL 46 to (50.48, 28.41, 27.28) mm, rotated rx -162.23 ry -14.17 rz 85.51 deg; joints [17.697, -60.279, 195.361, -43.826, 33.445, 48.788]
  MoveL 47 to (52.33, 29.24, 26.88) mm, rotated rx -159.24 ry -14.29 rz 84.65 deg; joints [19.605, -58.504, 193.723, -46.394, 36.564, 51.433]
  MoveL 48 to (52.74, 29.46, 26.78) mm, rotated rx -157.7 ry -14.43 rz 84.16 deg; joints [20.466, -57.44, 192.628, -47.265, 38.281, 52.259]
  MoveL 49 to (53.95, 30.22, 26.52) mm, rotated rx -156.91 ry -14.74 rz 83.81 deg; joints [20.976, -56.699, 191.717, -47.176, 39.439, 52.261]
  MoveL 50 to (54.91, 30.99, 26.37) mm, rotated rx -156.56 ry -15.6 rz 83.35 deg; joints [21.091, -55.764, 190.082, -45.61, 40.755, 50.742]
  MoveL 51 to (55.55, 31.66, 26.33) mm, rotated rx -156.68 ry -16.52 rz 83.01 deg; joints [20.897, -55.075, 188.6, -43.658, 41.69, 48.823]
  MoveL 52 to (55.83, 32.03, 26.35) mm, rotated rx -156.91 ry -17.25 rz 82.79 deg; joints [20.644, -54.584, 187.466, -42.07, 42.333, 47.238]
  MoveL 53 to (56.07, 32.4, 26.39) mm, rotated rx -157.15 ry -17.91 rz 82.62 deg; joints [20.395, -54.172, 186.481, -40.659, 42.891, 45.833]
  MoveL 54 to (56.3, 32.82, 26.46) mm, rotated rx -157.36 ry -18.59 rz 82.43 deg; joints [20.156, -53.721, 185.441, -39.267, 43.528, 44.445]
  MoveL 55 to (56.44, 33.14, 26.53) mm, rotated rx -157.51 ry -19.21 rz 82.24 deg; joints [19.952, -53.269, 184.457, -38.083, 44.159, 43.251]
  MoveL 56 to (56.56, 33.46, 26.62) mm, rotated rx -157.6 ry -19.77 rz 82.06 deg; joints [19.786, -52.83, 183.535, -37.066, 44.788, 42.223]
  MoveL 57 to (56.66, 33.79, 26.72) mm, rotated rx -157.64 ry -20.22 rz 81.91 deg; joints [19.669, -52.461, 182.774, -36.284, 45.339, 41.431]
  MoveL 58 to (56.68, 33.88, 26.75) mm, rotated rx -157.64 ry -20.7 rz 81.73 deg; joints [19.552, -51.995, 181.887, -35.519, 45.964, 40.636]
  MoveL 59 to (56.78, 34.53, 27.01) mm, rotated rx -157.53 ry -21.47 rz 81.39 deg; joints [19.438, -51.252, 180.475, -34.409, 47.097, 39.493]
  MoveL 60 to (56.77, 35.2, 27.32) mm, rotated rx -157.2 ry -22.41 rz 80.9 deg; joints [19.369, -50.193, 178.583, -33.27, 48.663, 38.282]
  MoveL 61 to (56.44, 35.96, 27.82) mm, rotated rx -156.61 ry -23.2 rz 80.33 deg; joints [19.426, -49.137, 176.796, -32.586, 50.281, 37.485]
  MoveL 62 to (56.18, 36.71, 28.31) mm, rotated rx -155.89 ry -23.77 rz 79.77 deg; joints [19.596, -48.198, 175.303, -32.309, 51.726, 37.104]
  MoveL 63 to (55.67, 37.62, 29) mm, rotated rx -155.33 ry -24.17 rz 79.35 deg; joints [19.721, -47.616, 174.341, -32.175, 52.775, 36.876]
  MoveL 64 to (55.04, 38.39, 29.67) mm, rotated rx -155.12 ry -24.42 rz 79.15 deg; joints [19.703, -47.432, 173.926, -31.984, 53.289, 36.617]
  MoveL 65 to (54.33, 39.06, 30.33) mm, rotated rx -155.52 ry -24.68 rz 79.24 deg; joints [19.404, -47.672, 173.981, -31.398, 53.243, 36.005]
  MoveL 66 to (53.29, 39.83, 31.17) mm, rotated rx -156.8 ry -25.03 rz 79.72 deg; joints [18.639, -48.462, 174.56, -30.046, 52.547, 34.662]
  MoveL 67 to (52.07, 40.53, 32) mm, rotated rx -158.54 ry -25.24 rz 80.49 deg; joints [17.671, -49.674, 175.721, -28.482, 51.281, 33.122]
  MoveL 68 to (51.54, 40.79, 32.31) mm, rotated rx -160.5 ry -25.46 rz 81.35 deg; joints [16.619, -50.737, 176.704, -26.585, 49.976, 31.29]
  MoveL 69 to (50, 41.45, 33.11) mm, rotated rx -163.38 ry -25.79 rz 82.6 deg; joints [14.952, -52.241, 178.072, -23.538, 48.225, 28.24]
  MoveL 70 to (48.35, 42.02, 33.8) mm, rotated rx -167.07 ry -25.95 rz 84.26 deg; joints [12.818, -54.05, 179.899, -19.469, 45.938, 24.152]
  MoveL 71 to (46.59, 42.52, 34.36) mm, rotated rx -170.66 ry -25.95 rz 85.88 deg; joints [10.659, -55.628, 181.601, -15.114, 43.863, 19.718]
  MoveL 72 to (45.48, 42.78, 34.62) mm, rotated rx -173.81 ry -25.87 rz 87.29 deg; joints [8.756, -56.746, 182.881, -10.931, 42.29, 15.475]
  MoveL 73 to (43.56, 43.15, 34.94) mm, rotated rx -176.72 ry -25.76 rz 88.57 deg; joints [6.862, -57.654, 183.989, -6.737, 41.068, 11.114]
  MoveL 74 to (41.55, 43.46, 35.15) mm, rotated rx -178.94 ry -25.58 rz 89.54 deg; joints [5.339, -58.299, 184.865, -3.357, 40.21, 7.539]
  MoveL 75 to (39.45, 43.69, 35.27) mm, rotated rx -179.95 ry -25.48 rz 89.98 deg; joints [4.5, -58.613, 185.319, -1.703, 39.83, 5.674]
  MoveL 76 to (37.93, 43.8, 35.32) mm, rotated rx 179.88 ry -25.44 rz 90.05 deg; joints [4.234, -58.721, 185.474, -1.393, 39.723, 5.212]
  MoveL 77 to (34.92, 43.89, 35.35) mm, rotated rx 180 ry -25.44 rz 90 deg; joints [3.961, -58.776, 185.549, -1.447, 39.708, 4.965]
  MoveL 78 to (31.9, 43.8, 35.32) mm, rotated rx -179.97 ry -25.46 rz 89.99 deg; joints [3.639, -58.775, 185.552, -1.373, 39.717, 4.588]
  MoveL 79 to (28.97, 43.56, 35.2) mm, rotated rx 179.22 ry -25.46 rz 90.33 deg; joints [2.818, -58.793, 185.606, 0.034, 39.631, 2.878]
  MoveL 80 to (26.66, 43.24, 34.99) mm, rotated rx 176.89 ry -25.43 rz 91.34 deg; joints [1.144, -58.792, 185.721, 3.873, 39.528, -1.217]
  MoveL 81 to (24.46, 42.82, 34.63) mm, rotated rx 175.33 ry -25.38 rz 92.01 deg; joints [-0.048, -58.674, 185.721, 6.471, 39.55, -4.055]
  Set speed (1000.0 mm/s)
  MoveL 82 to (24.46, 42.82, 34.63) mm, rotated rx 175.33 ry -25.38 rz 92.01 deg; joints [-0.048, -58.674, 185.721, 6.471, 39.55, -4.055]
  MoveL 83 to (17.81, -0.15, 124.68) mm, rotated rx 175.33 ry -25.38 rz 92.01 deg; joints [-0.74, -52.426, 159.243, 4.953, 59.743, -2.231]
